// TwinCAT 3 PLC project Main
// ProgramVersion: 3.1.4026.22
// libraries:
//   mobject-core, * (mobject)
//   Tc2_Standard, * (Beckhoff Automation GmbH)
//   Tc2_System, * (Beckhoff Automation GmbH)
//   Tc2_Utilities, * (Beckhoff Automation GmbH)
//   Tc3_JsonXml, * (Beckhoff Automation GmbH)
//   Tc3_Module, * (Beckhoff Automation GmbH)
//   TcUnit, * (www.tcunit.org)
// project tree:
//   mobject-collections/ MobjectCollectionsExample.TcPOU, MobjectCollectionsUnitTests.TcPOU
//   mobject-collections/Tests/ DictionaryForwardEnumerator_TestSuite.TcPOU, DictionaryKeyValueForwardEnumerator_TestSuite.TcPOU (not stored), Dictionary_TestSuite.TcPOU (not stored), LinkedListForwardEnumerator_TestSuite.TcPOU, LinkedList_TestSuite.TcPOU, OrderedDicKeyValueForwardEnumerator_TestSuite.TcPOU, OrderedDictionaryForwardEnumerator_TestSuite.TcPOU (not stored), OrderedDictionary_TestSuite.TcPOU (not stored), QueueForwardEnumerator_TestSuite.TcPOU, Queue_TestSuite.TcPOU (not stored), StackForwardEnumerator_TestSuite.TcPOU (not stored), Stack_TestSuite.TcPOU
//   mobject-collections/Tests/Mocks/EventHandlers/ CollectionChangedEventHandler.TcPOU, CollectionDisposedEventHandler.TcPOU (not stored), CollectionEventHandler.TcPOU (not stored), CollectionEventHandlerBase.TcPOU, KeyValueCollectionChangedEventHandler.TcPOU (not stored), KeyValueCollectionDisposedEventHandler.TcPOU, KeyValueCollectionEventHandler.TcPOU
//   mobject-converters/ MobjectConvertersUnitTests.TcPOU
//   mobject-converters/Tests/ BOOL_TO_TestSuite.TcPOU (not stored), BYTE_TO_TestSuite.TcPOU, DATE_TO_TestSuite.TcPOU, DINT_TO_TestSuite.TcPOU, DT_TO_TestSuite.TcPOU (not stored), DWORD_TO_TestSuite.TcPOU (not stored), INT_TO_TestSuite.TcPOU, LINT_TO_TestSuite.TcPOU, LREAL_TO_TestSuite.TcPOU, LWORD_TO_TestSuite.TcPOU, REAL_TO_TestSuite.TcPOU, SINT_TO_TestSuite.TcPOU (not stored), STRING_TO_TestSuite.TcPOU, TIME_TO_TestSuite.TcPOU, TOD_TO_TestSuite.TcPOU, UDINT_TO_TestSuite.TcPOU, UINT_TO_TestSuite.TcPOU (not stored), ULINT_TO_TestSuite.TcPOU, USINT_TO_TestSuite.TcPOU, WORD_TO_TestSuite.TcPOU (not stored)
//   mobject-datatypes/ MobjectDatatypesUnitTests.TcPOU (not stored)
//   mobject-datatypes/Tests/ AliasDatatype_TestSuite.TcPOU (not stored), Datatype_TestSuite.TcPOU (not stored), EnumDatatype_TestSuite.TcPOU, StructuredDatatype_TestSuite.TcPOU (not stored), _ArrayDatatype_1D_TestSuite.TcPOU, _ArrayDatatype_2D_TestSuite.TcPOU, _ArrayDatatype_3D_TestSuite.TcPOU, _BIT_UsingMockStructure_TestSuite.TcPOU, _BOOL_TestSuite.TcPOU (not stored), _BYTE_TestSuite.TcPOU (not stored), _DINT_TestSuite.TcPOU, _DT_TestSuite.TcPOU (not stored), _DWORD_TestSuite.TcPOU (not stored), _INT_TestSuite.TcPOU (not stored), _LINT_TestSuite.TcPOU, _LREAL_TestSuite.TcPOU (not stored), _LWORD_TestSuite.TcPOU (not stored), _REAL_TestSuite.TcPOU, _SINT_TestSuite.TcPOU, _STRING_TestSuite.TcPOU (not stored), _TIME_OF_DAY_TestSuite.TcPOU (not stored), _TOD_TestSuite.TcPOU (not stored), _UDINT_TestSuite.TcPOU, _UINT_TestSuite.TcPOU, _ULINT_TestSuite.TcPOU, _USINT_TestSuite.TcPOU (not stored), _WORD_TestSuite.TcPOU (not stored)
//   mobject-datatypes/Tests/Mocks/1DimArray/ _Array0to10OfBool.TcPOU
//   mobject-datatypes/Tests/Mocks/2DimArray/ _Array0to1_0to2OfBool.TcPOU
//   mobject-datatypes/Tests/Mocks/3DimArray/ _Array0to1_0to2_0to3OfBool.TcPOU (not stored)
//   mobject-datatypes/Tests/Mocks/DUT/ MyStruct.TcDUT
//   mobject-datatypes/Tests/Mocks/ MockAliasDatatype_HRESULT.TcPOU, MockDatatype_BOOL.TcPOU (not stored), MockEnumDatatype_E_TcEventClass.TcPOU, MockStructuredDatatype_TIMESTRUCT.TcPOU, _MyStruct.TcPOU
//   mobject-deserialization/ MobjectDeserializationUnitTests.TcPOU (not stored)
//   mobject-deserialization/Tests/ CustomDeserializationFailedError_TestSuite.TcPOU, DeserializationErrorFactory_TestSuite.TcPOU, DeserializerGarbageCollector_TestSuite.TcPOU (not stored), IncorrectKeyTypeDeserializationError_TestSuite.TcPOU, IncorrectTypeDeserializationError_TestSuite.TcPOU, InvalidKeyDeserializationError_TestSuite.TcPOU, MissingKeyDeserializationError_TestSuite.TcPOU (not stored), InvalidArrayIndexDeserializationError_TestSuite.TcPOU (not stored)
//   mobject-deserialization/Tests/Mocks/ MockDisposableDeserializer.TcPOU
//   mobject-disposable/ MobjectDisposableUnitTests.TcPOU
//   mobject-disposable/Tests/ Disposable_TestSuite.TcPOU (not stored)
//   mobject-disposable/Tests/Mocks/ MockDisposable.TcPOU (not stored)
//   mobject-errors/ MobjectErrorsUnitTests.TcPOU
//   mobject-errors/Tests/ Error_TestSuite.TcPOU (not stored), NullError_TestSuite.TcPOU (not stored)
//   mobject-events/ MobjectEventsUnitTests.TcPOU
//   mobject-events/Tests/ EventEmitterInterface_TestSuite.TcPOU (not stored), EventEmitter_TestSuite.TcPOU (not stored), EventHandlerInterface_TestSuite.TcPOU (not stored), EventTargetInterface_TestSuite.TcPOU
//   mobject-events/Tests/Mocks/ MockEvent.TcPOU (not stored), MockEventHandler.TcPOU (not stored)
//   mobject-json/ MobjectJsonUnitTests.TcPOU
//   mobject-json/Tests/ JsonDeserializerArrayForwardEnumerator_TestSuite.TcPOU, JsonDeserializerObjectForwardEnumerator_TestSuite.TcPOU (not stored), JsonDeserializer_TestSuite.TcPOU, JsonDomParser_TestSuite.TcPOU, JsonSerializer_TestSuite.TcPOU
//   mobject-json/Tests/Mocks/ MockDeserializableUserObject.TcPOU, MockSerializableArray.TcPOU (not stored), MockSerializableUserObject.TcPOU
//   mobject-server/ MobjectServerUnitTests.TcPOU, Server_IntegrationTestSuite.TcPOU
//   mobject-server/Mocks/ AdjustableSizeReplyRpcHandler.TcPOU, RejectWithMessageAsyncHandler.TcPOU, RejectWithMessageSyncHandler.TcPOU, SyncToAsyncEchoRpcHandler.TcPOU
//   mobject-server/_Internal/ AsyncResponseSessionData_TestSuite.TcPOU, ChunkedRequestData_TestSuite.TcPOU
//   / PlcTask.TcTTO
//   Main/ MAIN.TcPOU
//   SharedMocks/ MockError.TcPOU, MockErrorVisitor.TcPOU (not stored), MockJsonSerializer.TcPOU
// real-time tasks:
//   TASK PlcTask: cycle T#10ms, priority 20, ADS port 350

CONFIGURATION Main
    RESOURCE PLC ON TwinCAT3
        TASK PlcTask(INTERVAL := T#10ms, PRIORITY := 20);
        PROGRAM MAIN WITH PlcTask : MAIN;
    END_RESOURCE
END_CONFIGURATION

// ---- mobject-datatypes/Tests/Mocks/DUT/MyStruct.TcDUT
TYPE MyStruct :
STRUCT
	MyBit : BIT;
END_STRUCT
END_TYPE

// ---- Main/MAIN.TcPOU
PROGRAM MAIN
VAR
END_VAR

// unit tests
MobjectCollectionsUnitTests();
MobjectConvertersUnitTests();
MobjectDatatypesUnitTests();
MobjectDeserializationUnitTests();
MobjectDisposableUnitTests();
MobjectErrorsUnitTests();
MobjectEventsUnitTests();
MobjectJsonUnitTests();
MobjectServerUnitTests();

// examples
MobjectCollectionsExample();

// tcunit
TcUnit.RUN();

END_PROGRAM

// ---- mobject-collections/MobjectCollectionsUnitTests.TcPOU
PROGRAM MobjectCollectionsUnitTests
VAR
	dictionary_TestSuite : Dictionary_TestSuite;
	dictionaryForwardEnumerator_TestSuite : DictionaryForwardEnumerator_TestSuite;
	dictionaryKeyValueForwardEnumerator_TestSuite : DictionaryKeyValueForwardEnumerator_TestSuite;
	orderedDictionary_TestSuite : OrderedDictionary_TestSuite;
	orderedDictionaryForwardEnumerator_TestSuite : OrderedDictionaryForwardEnumerator_TestSuite;
	orderedDicKeyValueForwardEnumerator_TestSuite : OrderedDicKeyValueForwardEnumerator_TestSuite;
    linkedList_TestSuite : LinkedList_TestSuite;
	linkedListForwardEnumerator_TestSuite : LinkedListForwardEnumerator_TestSuite;
	queue_TestSuite : Queue_TestSuite;
	queueForwardEnumerator_TestSuite : QueueForwardEnumerator_TestSuite;
    stack_TestSuite : Stack_TestSuite;
	stackForwardEnumerator_TestSuite : StackForwardEnumerator_TestSuite;
END_VAR

END_PROGRAM

// ---- mobject-collections/Tests/DictionaryForwardEnumerator_TestSuite.TcPOU
FUNCTION_BLOCK DictionaryForwardEnumerator_TestSuite EXTENDS TcUnit.FB_TestSuite
VAR
END_VAR

CheckIsValidAtStart();
CheckMoveNextReturnsFalseAtTheEnd();
CheckMoveNextReturnsTrueSingleItem();
CheckMoveNextReturnsFalseWhenEmpty();
CheckMoveNextReturnsTrueMultipleItems();
CheckReset();
CheckTryGet();
CheckTryGetTo();
CheckWorksWithArrays();
CheckWorksWithIntegers();
CheckWorksWithStrings();

METHOD PRIVATE CheckIsValidAtStart
VAR
	result : BOOL;
	dictionary : Dictionary;
	enumerator : I_ForwardEnumerator;
END_VAR
TEST('CheckIsValidAtStart');

enumerator := dictionary.GetEnumerator();

result := enumerator.IsValid;
enumerator.Dispose();

AssertTrue(
	Condition := result,
	Message := 'IsValid returned false'
);

TEST_FINISHED();
END_METHOD

METHOD PRIVATE CheckMoveNextReturnsFalseAtTheEnd
VAR
	in1 : INT := 123;
	result : BOOL;
	dictionary : Dictionary;
	enumerator : I_ForwardEnumerator;
END_VAR
TEST('CheckMoveNextReturnsFalseAtTheEnd');

dictionary.TryAdd('a',in1);
enumerator := dictionary.GetEnumerator();

enumerator.MoveNext();
result := enumerator.MoveNext();

enumerator.Dispose();

AssertFalse(result,
    'MoveNext did not correctly signal the end of the enumeration');
	
TEST_FINISHED();
END_METHOD

METHOD PRIVATE CheckMoveNextReturnsFalseWhenEmpty
VAR
	result : BOOL;
	dictionary : Dictionary;
	enumerator : I_ForwardEnumerator;
	count : DINT;
END_VAR
TEST('CheckMoveNextReturnsFalseWhenEmpty');

count := dictionary.Count;
enumerator := dictionary.GetEnumerator();

result := enumerator.MoveNext();
enumerator.Dispose();

AssertFalse(Condition := result,
    Message := 'MoveNext did not correctly signal the end of the enumeration');

TEST_FINISHED();
END_METHOD

METHOD PRIVATE CheckMoveNextReturnsTrueMultipleItems
VAR
	in1 : INT := 123;
	in2 : INT := 456;
	in3 : INT := 789;
	result : BOOL;
	dictionary : Dictionary;
	enumerator : I_ForwardEnumerator;
END_VAR
TEST('CheckMoveNextReturnsTrueMultipleItems');

dictionary.TryAdd('a',in1);
dictionary.TryAdd('b',in2);
dictionary.TryAdd('c',in3);
enumerator := dictionary.GetEnumerator();

result := enumerator.MoveNext();
enumerator.Dispose();

AssertTrue(result, 'MoveNext did not correctly signal there were more items to follow');

TEST_FINISHED();
END_METHOD

METHOD PRIVATE CheckMoveNextReturnsTrueSingleItem
VAR
	in1 : INT := 123;
	result : BOOL;
	dictionary : Dictionary;
	enumerator : I_ForwardEnumerator;
END_VAR
TEST('CheckMoveNextReturnsTrueSingleItem');

dictionary.TryAdd('a',in1);
enumerator := dictionary.GetEnumerator();

result := enumerator.MoveNext();
enumerator.Dispose();

AssertTrue(result,
    'MoveNext did not correctly signal there were more items to follow');
	
TEST_FINISHED();
END_METHOD

METHOD PRIVATE CheckReset
VAR
	in1 : ARRAY [0..1] OF REAL := [0.1,2.3];
	in2 : ARRAY [0..1] OF REAL := [1.2,3.4];
	in3 : ARRAY [0..1] OF REAL := [2.3,4.5];
	out : ARRAY [0..1] OF REAL;
	expected : ARRAY [0..1] OF REAL := [0.1,2.3];
	dictionary : Dictionary;
	enumerator : I_ForwardEnumerator;
END_VAR
TEST('CheckReset');

dictionary.TryAdd('a',in1);
dictionary.TryAdd('b',in2);
dictionary.TryAdd('c',in3);

enumerator := dictionary.GetEnumerator();

enumerator.MoveNext();
enumerator.MoveNext();
enumerator.Reset();
enumerator.MoveNext();
enumerator.TryGet(out);

enumerator.Dispose();

AssertEquals(
	Expected := expected,
	Actual := out,
	Message := 'Did not produce the expected result'
);

TEST_FINISHED();
END_METHOD

METHOD PRIVATE CheckTryGet
VAR
	in : INT := 123;
	out : INT;
	expected : INT := 123;
	result : BOOL;
	dictionary : Dictionary;
	enumerator : I_ForwardEnumerator;
END_VAR
TEST('CheckTryGet');

dictionary.TryAdd('a',in);
enumerator := dictionary.GetEnumerator();
enumerator.MoveNext();

result := enumerator.TryGet(out);
enumerator.Dispose();

AssertTrue(
	Condition := result,
	Message := 'Method returned false'
);

AssertEquals(
	Expected := expected,
	Actual := out,
	Message := 'Did not produce the expected result'
);

TEST_FINISHED();
END_METHOD

METHOD PRIVATE CheckTryGetTo
VAR
	in : INT := 123;
	out : INT;
	expected : INT := 123;
	result : BOOL;
	dictionary : Dictionary;
	enumerator : I_ForwardEnumerator;
END_VAR
TEST('CheckTryGetTo');

dictionary.TryAdd('a',in);
enumerator := dictionary.GetEnumerator();
enumerator.MoveNext();

result := enumerator.TryGetTo(ADR(out),SIZEOF(out));
enumerator.Dispose();

AssertTrue(
	Condition := result,
	Message := 'Method returned false'
);

AssertEquals(
	Expected := expected,
	Actual := out,
	Message := 'Did not produce the expected result'
);

TEST_FINISHED();
END_METHOD

METHOD PRIVATE CheckWorksWithArrays
VAR
	in1 : ARRAY [0..1] OF REAL := [0.1,2.3];
	in2 : ARRAY [0..1] OF REAL := [1.2,3.4];
	in3 : ARRAY [0..1] OF REAL := [2.3,4.5];
	out1 : ARRAY [0..1] OF REAL;
	out2 : ARRAY [0..1] OF REAL;
	out3 : ARRAY [0..1] OF REAL;
	expected1 : ARRAY [0..1] OF REAL := [0.1,2.3];
	expected2 : ARRAY [0..1] OF REAL := [1.2,3.4];
	expected3 : ARRAY [0..1] OF REAL := [2.3,4.5];
	dictionary : Dictionary;
	enumerator : I_ForwardEnumerator;
END_VAR
TEST('CheckWorksWithArrays');

dictionary.TryAdd('c',in3);
dictionary.TryAdd('b',in2);
dictionary.TryAdd('a',in1);

enumerator := dictionary.GetEnumerator();

enumerator.MoveNext();
enumerator.TryGet(out1);
enumerator.MoveNext();
enumerator.TryGet(out2);
enumerator.MoveNext();
enumerator.TryGet(out3);

enumerator.Dispose();

AssertEquals(
	Expected := expected1,
	Actual := out1,
	Message := 'Did not produce the expected 1st result'
);

AssertEquals(
	Expected := expected2,
	Actual := out2,
	Message := 'Did not produce the expected 2nd result'
);

AssertEquals(
	Expected := expected3,
	Actual := out3,
	Message := 'Did not produce the expected 3rd result'
);

TEST_FINISHED();
END_METHOD

METHOD PRIVATE CheckWorksWithIntegers
VAR
	in1 : INT := 123;
	in2 : INT := 234;
	in3 : INT := 345;
	out1 : INT;
	out2 : INT;
	out3 : INT;
	expected1 : INT := 123;
	expected2 : INT := 234;
	expected3 : INT := 345;
	dictionary : Dictionary;
	enumerator : I_ForwardEnumerator;
END_VAR
TEST('CheckWorksWithIntegers');

dictionary.TryAdd('c',in3);
dictionary.TryAdd('b',in2);
dictionary.TryAdd('a',in1);

enumerator := dictionary.GetEnumerator();

enumerator.MoveNext();
enumerator.TryGet(out1);
enumerator.MoveNext();
enumerator.TryGet(out2);
enumerator.MoveNext();
enumerator.TryGet(out3);

enumerator.Dispose();

AssertEquals(
	Expected := expected1,
	Actual := out1,
	Message := 'Did not produce the expected 1st result'
);

AssertEquals(
	Expected := expected2,
	Actual := out2,
	Message := 'Did not produce the expected 2nd result'
);

AssertEquals(
	Expected := expected3,
	Actual := out3,
	Message := 'Did not produce the expected 3rd result'
);

TEST_FINISHED();
END_METHOD

METHOD PRIVATE CheckWorksWithStrings
VAR
	in1 : STRING := 'test1';
	in2 : STRING := 'test2';
	in3 : STRING := 'test3';
	out1 : STRING;
	out2 : STRING;
	out3 : STRING;
	expected1 : STRING := 'test1';
	expected2 : STRING := 'test2';
	expected3 : STRING := 'test3';
	dictionary : Dictionary;
	enumerator : I_ForwardEnumerator;
END_VAR
TEST('CheckWorksWithStrings');

dictionary.TryAdd('c',in3);
dictionary.TryAdd('b',in2);
dictionary.TryAdd('a',in1);

enumerator := dictionary.GetEnumerator();

enumerator.MoveNext();
enumerator.TryGet(out1);
enumerator.MoveNext();
enumerator.TryGet(out2);
enumerator.MoveNext();
enumerator.TryGet(out3);

enumerator.Dispose();

AssertEquals(
	Expected := expected1,
	Actual := out1,
	Message := 'Did not produce the expected 1st result'
);

AssertEquals(
	Expected := expected2,
	Actual := out2,
	Message := 'Did not produce the expected 2nd result'
);

AssertEquals(
	Expected := expected3,
	Actual := out3,
	Message := 'Did not produce the expected 3rd result'
);

TEST_FINISHED();
END_METHOD

END_FUNCTION_BLOCK

// ---- mobject-collections/Tests/OrderedDicKeyValueForwardEnumerator_TestSuite.TcPOU
FUNCTION_BLOCK OrderedDicKeyValueForwardEnumerator_TestSuite EXTENDS TcUnit.FB_TestSuite
VAR
END_VAR

CheckIsValidAtStart();
CheckKey();
CheckMoveNextReturnsFalseAtTheEnd();
CheckMoveNextReturnsTrueSingleItem();
CheckMoveNextReturnsFalseWhenEmpty();
CheckMoveNextReturnsTrueMultipleItems();
CheckReset();
CheckTryGet();
CheckTryGetTo();
CheckWorksWithArrays();
CheckWorksWithIntegers();
CheckWorksWithStrings();

METHOD PRIVATE CheckIsValidAtStart
VAR
	result : BOOL;
	dictionary : OrderedDictionary;
	enumerator : I_KeyValueForwardEnumerator;
END_VAR
TEST('CheckIsValidAtStart');

enumerator := dictionary.GetKeyValueEnumerator();

result := enumerator.IsValid;
enumerator.Dispose();

AssertTrue(
	Condition := result,
	Message := 'IsValid returned false'
);

TEST_FINISHED();
END_METHOD

METHOD PRIVATE CheckKey
VAR
	in1 : STRING := 'test1';
	in2 : STRING := 'test2';
	in3 : STRING := 'test3';
	out1 : STRING;
	out2 : STRING;
	out3 : STRING;
	expected1 : STRING := 'a';
	expected2 : STRING := 'b';
	expected3 : STRING := 'c';
	dictionary : OrderedDictionary;
	enumerator : I_KeyValueForwardEnumerator;
END_VAR
TEST('CheckKey');

dictionary.TryAdd('a',in1);
dictionary.TryAdd('b',in2);
dictionary.TryAdd('c',in3);

enumerator := dictionary.GetKeyValueEnumerator();

enumerator.MoveNext();
out1 := enumerator.Key;
enumerator.MoveNext();
out2 := enumerator.Key;
enumerator.MoveNext();
out3 := enumerator.Key;

enumerator.Dispose();

AssertEquals(
	Expected := expected1,
	Actual := out1,
	Message := 'Did not produce the expected 1st key'
);

AssertEquals(
	Expected := expected2,
	Actual := out2,
	Message := 'Did not produce the expected 2nd key'
);

AssertEquals(
	Expected := expected3,
	Actual := out3,
	Message := 'Did not produce the expected 3rd key'
);

TEST_FINISHED();
END_METHOD

METHOD PRIVATE CheckMoveNextReturnsFalseAtTheEnd
VAR
	in1 : INT := 123;
	result : BOOL;
	dictionary : OrderedDictionary;
	enumerator : I_KeyValueForwardEnumerator;
END_VAR
TEST('CheckMoveNextReturnsFalseAtTheEnd');

dictionary.TryAdd('a',in1);
enumerator := dictionary.GetKeyValueEnumerator();

enumerator.MoveNext();
result := enumerator.MoveNext();

enumerator.Dispose();

AssertFalse(result,
    'MoveNext did not correctly signal the end of the enumeration');
	
TEST_FINISHED();
END_METHOD

METHOD PRIVATE CheckMoveNextReturnsFalseWhenEmpty
VAR
	result : BOOL;
	dictionary : OrderedDictionary;
	enumerator : I_KeyValueForwardEnumerator;
	count : DINT;
END_VAR
TEST('CheckMoveNextReturnsFalseWhenEmpty');

count := dictionary.Count;
enumerator := dictionary.GetKeyValueEnumerator();

result := enumerator.MoveNext();
enumerator.Dispose();

AssertFalse(Condition := result,
    Message := 'MoveNext did not correctly signal the end of the enumeration');

TEST_FINISHED();
END_METHOD

METHOD PRIVATE CheckMoveNextReturnsTrueMultipleItems
VAR
	in1 : INT := 123;
	in2 : INT := 456;
	in3 : INT := 789;
	result : BOOL;
	dictionary : OrderedDictionary;
	enumerator : I_KeyValueForwardEnumerator;
END_VAR
TEST('CheckMoveNextReturnsTrueMultipleItems');

dictionary.TryAdd('a',in1);
dictionary.TryAdd('b',in2);
dictionary.TryAdd('c',in3);
enumerator := dictionary.GetKeyValueEnumerator();

result := enumerator.MoveNext();
enumerator.Dispose();

AssertTrue(result, 'MoveNext did not correctly signal there were more items to follow');

TEST_FINISHED();
END_METHOD

METHOD PRIVATE CheckMoveNextReturnsTrueSingleItem
VAR
	in1 : INT := 123;
	result : BOOL;
	dictionary : OrderedDictionary;
	enumerator : I_KeyValueForwardEnumerator;
END_VAR
TEST('CheckMoveNextReturnsTrueSingleItem');

dictionary.TryAdd('a',in1);
enumerator := dictionary.GetKeyValueEnumerator();

result := enumerator.MoveNext();
enumerator.Dispose();

AssertTrue(result,
    'MoveNext did not correctly signal there were more items to follow');
	
TEST_FINISHED();
END_METHOD

METHOD PRIVATE CheckReset
VAR
	in1 : ARRAY [0..1] OF REAL := [0.1,2.3];
	in2 : ARRAY [0..1] OF REAL := [1.2,3.4];
	in3 : ARRAY [0..1] OF REAL := [2.3,4.5];
	out : ARRAY [0..1] OF REAL;
	expected : ARRAY [0..1] OF REAL := [0.1,2.3];
	dictionary : OrderedDictionary;
	enumerator : I_KeyValueForwardEnumerator;
END_VAR
TEST('CheckReset');

dictionary.TryAdd('a',in1);
dictionary.TryAdd('b',in2);
dictionary.TryAdd('c',in3);

enumerator := dictionary.GetKeyValueEnumerator();

enumerator.MoveNext();
enumerator.MoveNext();
enumerator.Reset();
enumerator.MoveNext();
enumerator.TryGet(out);

enumerator.Dispose();

AssertEquals(
	Expected := expected,
	Actual := out,
	Message := 'Did not produce the expected result'
);

TEST_FINISHED();
END_METHOD

METHOD PRIVATE CheckTryGet
VAR
	in : INT := 123;
	out : INT;
	expected : INT := 123;
	result : BOOL;
	dictionary : OrderedDictionary;
	enumerator : I_KeyValueForwardEnumerator;
END_VAR
TEST('CheckTryGet');

dictionary.TryAdd('a',in);
enumerator := dictionary.GetKeyValueEnumerator();
enumerator.MoveNext();

result := enumerator.TryGet(out);
enumerator.Dispose();

AssertTrue(
	Condition := result,
	Message := 'Method returned false'
);

AssertEquals(
	Expected := expected,
	Actual := out,
	Message := 'Did not produce the expected result'
);

TEST_FINISHED();
END_METHOD

METHOD PRIVATE CheckTryGetTo
VAR
	in : INT := 123;
	out : INT;
	expected : INT := 123;
	result : BOOL;
	dictionary : OrderedDictionary;
	enumerator : I_KeyValueForwardEnumerator;
END_VAR
TEST('CheckTryGetTo');

dictionary.TryAdd('a',in);
enumerator := dictionary.GetKeyValueEnumerator();
enumerator.MoveNext();

result := enumerator.TryGetTo(ADR(out),SIZEOF(out));
enumerator.Dispose();

AssertTrue(
	Condition := result,
	Message := 'Method returned false'
);

AssertEquals(
	Expected := expected,
	Actual := out,
	Message := 'Did not produce the expected result'
);

TEST_FINISHED();
END_METHOD

METHOD PRIVATE CheckWorksWithArrays
VAR
	in1 : ARRAY [0..1] OF REAL := [0.1,2.3];
	in2 : ARRAY [0..1] OF REAL := [1.2,3.4];
	in3 : ARRAY [0..1] OF REAL := [2.3,4.5];
	out1 : ARRAY [0..1] OF REAL;
	out2 : ARRAY [0..1] OF REAL;
	out3 : ARRAY [0..1] OF REAL;
	expected1 : ARRAY [0..1] OF REAL := [0.1,2.3];
	expected2 : ARRAY [0..1] OF REAL := [1.2,3.4];
	expected3 : ARRAY [0..1] OF REAL := [2.3,4.5];
	dictionary : OrderedDictionary;
	enumerator : I_KeyValueForwardEnumerator;
END_VAR
TEST('CheckWorksWithArrays');

dictionary.TryAdd('c',in1);
dictionary.TryAdd('b',in2);
dictionary.TryAdd('a',in3);

enumerator := dictionary.GetKeyValueEnumerator();

enumerator.MoveNext();
enumerator.TryGet(out1);
enumerator.MoveNext();
enumerator.TryGet(out2);
enumerator.MoveNext();
enumerator.TryGet(out3);

enumerator.Dispose();

AssertEquals(
	Expected := expected1,
	Actual := out1,
	Message := 'Did not produce the expected 1st result'
);

AssertEquals(
	Expected := expected2,
	Actual := out2,
	Message := 'Did not produce the expected 2nd result'
);

AssertEquals(
	Expected := expected3,
	Actual := out3,
	Message := 'Did not produce the expected 3rd result'
);

TEST_FINISHED();
END_METHOD

METHOD PRIVATE CheckWorksWithIntegers
VAR
	in1 : INT := 123;
	in2 : INT := 234;
	in3 : INT := 345;
	out1 : INT;
	out2 : INT;
	out3 : INT;
	expected1 : INT := 123;
	expected2 : INT := 234;
	expected3 : INT := 345;
	dictionary : OrderedDictionary;
	enumerator : I_KeyValueForwardEnumerator;
END_VAR
TEST('CheckWorksWithIntegers');

dictionary.TryAdd('c',in1);
dictionary.TryAdd('b',in2);
dictionary.TryAdd('a',in3);

enumerator := dictionary.GetKeyValueEnumerator();

enumerator.MoveNext();
enumerator.TryGet(out1);
enumerator.MoveNext();
enumerator.TryGet(out2);
enumerator.MoveNext();
enumerator.TryGet(out3);

enumerator.Dispose();

AssertEquals(
	Expected := expected1,
	Actual := out1,
	Message := 'Did not produce the expected 1st result'
);

AssertEquals(
	Expected := expected2,
	Actual := out2,
	Message := 'Did not produce the expected 2nd result'
);

AssertEquals(
	Expected := expected3,
	Actual := out3,
	Message := 'Did not produce the expected 3rd result'
);

TEST_FINISHED();
END_METHOD

METHOD PRIVATE CheckWorksWithStrings
VAR
	in1 : STRING := 'test1';
	in2 : STRING := 'test2';
	in3 : STRING := 'test3';
	out1 : STRING;
	out2 : STRING;
	out3 : STRING;
	expected1 : STRING := 'test1';
	expected2 : STRING := 'test2';
	expected3 : STRING := 'test3';
	dictionary : OrderedDictionary;
	enumerator : I_KeyValueForwardEnumerator;
END_VAR
TEST('CheckWorksWithStrings');

dictionary.TryAdd('c',in1);
dictionary.TryAdd('b',in2);
dictionary.TryAdd('a',in3);

enumerator := dictionary.GetKeyValueEnumerator();

enumerator.MoveNext();
enumerator.TryGet(out1);
enumerator.MoveNext();
enumerator.TryGet(out2);
enumerator.MoveNext();
enumerator.TryGet(out3);

enumerator.Dispose();

AssertEquals(
	Expected := expected1,
	Actual := out1,
	Message := 'Did not produce the expected 1st result'
);

AssertEquals(
	Expected := expected2,
	Actual := out2,
	Message := 'Did not produce the expected 2nd result'
);

AssertEquals(
	Expected := expected3,
	Actual := out3,
	Message := 'Did not produce the expected 3rd result'
);

TEST_FINISHED();
END_METHOD

END_FUNCTION_BLOCK

// ---- mobject-collections/Tests/LinkedList_TestSuite.TcPOU
FUNCTION_BLOCK PUBLIC LinkedList_TestSuite EXTENDS TcUnit.FB_TestSuite

// check datatypes are handled correctly
CheckListWorksWithIntegers();
CheckListWorksWithStrings();
CheckListWorksWithArrays();

// all other checks
CheckLinkedListImplementsI_LinkedList();
CheckFirstIsCorrectWithOneValue();
CheckFirstIsCorrectWithMultipleValues();
CheckLastIsCorrectWithOneValue();
CheckLastIsCorrectWithMultipleValues();
CheckAddAfter();
CheckAddBefore();
CheckAddFirst();
CheckAddItem();
CheckAddLast();
CheckClear();
CheckRemove();
CheckRemoveFirst();
CheckTryRemoveItem();
CheckRemoveLast();
CheckCount();
CheckFind();
CheckFindLast();
CheckLinkedListReturnsEnumerator();
CheckOnChangedEvent();
CheckOnDisposedEvent();
CheckOnceEvent();
CheckOffEvent();
CheckTryCopyTo();
CheckEnumeratorIsInvalidAfterChange();
CheckIsEmptyWhenEmpty();
CheckIsEmptyWhenFull();

METHOD PUBLIC CheckAddAfter
VAR
	in1 : INT := 123;
	in2 : INT := 456;
	in3 : INT := 789;
	out : INT;
	expected : INT := 789;
	linkedList : LinkedList;
END_VAR
TEST('CheckAddAfter');

// @TEST-FIXTURE
linkedList.AddFirst(in1); // (first->) 123 (<-last)
linkedList.AddFirst(in2); // (first->) 456, 123 (<-last)

// @TEST-RUN
linkedList.AddAfter(linkedList.Last, in3); // (first->) 456, 123, 789 (<-last)
linkedList.Last.TryGet(out);

// @TEST-ASSSERT
AssertEquals(
	Expected := expected,
	Actual := out,
	Message := 'Did not produce the expected result'
);

TEST_FINISHED();
END_METHOD

METHOD PUBLIC CheckAddBefore
VAR
	in1 : INT := 123;
	in2 : INT := 456;
	in3 : INT := 789;
	out : INT;
	expected : INT := 789;
	linkedList : LinkedList;
END_VAR
TEST('CheckAddBefore');

// @TEST-FIXTURE
linkedList.AddFirst(in1); // (first->) 123 (<-last)
linkedList.AddFirst(in2); // (first->) 456, 123 (<-last)

// @TEST-RUN
linkedList.AddBefore(linkedList.First, in3); // (first->) 789, 456, 123 (<-last)
linkedList.First.TryGet(out);

// @TEST-ASSSERT
AssertEquals(
	Expected := expected,
	Actual := out,
	Message := 'Did not produce the expected result'
);

TEST_FINISHED();
END_METHOD

METHOD PUBLIC CheckAddFirst
VAR
	in1 : INT := 123;
	in2 : INT := 456;
	in3 : INT := 789;
	out : INT;
	expected : INT := 789;
	linkedList : LinkedList;
END_VAR
TEST('CheckAddFirst');

// @TEST-FIXTURE
linkedList.AddLast(in1); // (first->) 123 (<-last)
linkedList.AddLast(in2); // (first->) 123, 456 (<-last)

// @TEST-RUN
linkedList.AddFirst(in3); // (first->) 789, 123, 456 (<-last)
linkedList.First.TryGet(out);

// @TEST-ASSSERT
AssertEquals(
	Expected := expected,
	Actual := out,
	Message := 'Did not produce the expected result'
);

TEST_FINISHED();
END_METHOD

METHOD PUBLIC CheckAddItem
VAR
	in1 : INT := 123;
	in2 : INT := 456;
	in3 : INT := 789;
	out : INT;
	expected : INT := 789;
	linkedList : LinkedList;
END_VAR
TEST('CheckAddItem');

// @TEST-FIXTURE
linkedList.AddFirst(in1); // (first->) 123 (<-last)
linkedList.AddFirst(in2); // (first->) 456, 123 (<-last)

// @TEST-RUN
linkedList.AddItem(in3); // (first->) 456, 123, 789 (<-last)
linkedList.Last.TryGet(out);

// @TEST-ASSSERT
AssertEquals(
	Expected := expected,
	Actual := out,
	Message := 'Did not produce the expected result'
);

TEST_FINISHED();
END_METHOD

METHOD PUBLIC CheckAddLast
VAR
	in1 : INT := 123;
	in2 : INT := 456;
	in3 : INT := 789;
	out : INT;
	expected : INT := 789;
	linkedList : LinkedList;
END_VAR
TEST('CheckAddLast');

// @TEST-FIXTURE
linkedList.AddFirst(in1); // (first->) 123 (<-last)
linkedList.AddFirst(in2); // (first->) 456, 123 (<-last)

// @TEST-RUN
linkedList.AddLast(in3); // (first->) 456, 123, 789 (<-last)
linkedList.Last.TryGet(out);

// @TEST-ASSSERT
AssertEquals(
	Expected := expected,
	Actual := out,
	Message := 'Did not produce the expected result'
);

TEST_FINISHED();
END_METHOD

METHOD PUBLIC CheckClear
VAR
	in1 : INT := 123;
	in2 : INT := 456;
	out : INT;
	expected : INT := 456;
	linkedList : LinkedList;
END_VAR
TEST('CheckClear');

// @TEST-FIXTURE
linkedList.AddFirst(in1); // (first->) 123 (<-last)

// @TEST-RUN
linkedList.Clear();
linkedList.AddFirst(in2); // (first->) 456 (<-last) // if clear did not work then it would have (first->) 456, 123 (<-last)
linkedList.Last.TryGet(out);

// @TEST-ASSSERT
AssertEquals(
	Expected := expected,
	Actual := out,
	Message := 'Did not produce the expected result'
);

TEST_FINISHED();
END_METHOD

METHOD PUBLIC CheckCount
VAR
	in1 : INT := 123;
	in2 : INT := 456;
	in3 : INT := 789;
	out : DINT;
	expected : DINT := 3;
	linkedList : LinkedList;
END_VAR
TEST('CheckCount');

// @TEST-FIXTURE
linkedList.AddFirst(in1);
linkedList.AddFirst(in2);
linkedList.AddFirst(in3);

// @TEST-RUN
out := linkedList.Count;

// @TEST-ASSSERT
AssertEquals(
	Expected := expected,
	Actual := out,
	Message := 'Did not produce the expected result'
);

TEST_FINISHED();
END_METHOD

METHOD PUBLIC CheckEnumeratorIsInvalidAfterChange
VAR
	in : INT := 123;
	result : BOOL;
	linkedList : LinkedList;
	enumerator : I_ForwardEnumerator;
END_VAR
TEST('CheckEnumeratorIsInvalidAfterChange');

// @TEST-FIXTURE
enumerator := linkedList.GetEnumerator();
linkedList.AddItem(in);

// @TEST-RUN
result := enumerator.IsValid;
enumerator.Dispose();

// @TEST-ASSSERT
AssertFalse(
	Condition := result,
	Message := 'Method returned true'
);

TEST_FINISHED();
END_METHOD

METHOD PUBLIC CheckFind
VAR
	in1 : INT := 123;
	in2 : INT := 456;
	foundNode : I_LinkedListNode;
	linkedList : LinkedList;
END_VAR
TEST('CheckFind');

// @TEST-FIXTURE
linkedList.AddFirst(in1); // (first->) 123 (<-last)
linkedList.AddFirst(in2); // (first->) 456, 123 (<-last)
linkedList.AddFirst(in1); // (first->) 123, 456, 123 (<-last)

// @TEST-RUN
foundNode := linkedList.Find(in1);

// @TEST-ASSSERT
AssertTrue(
	Condition := (foundNode = linkedList.First),
	Message := 'Did find the correct node'
);

TEST_FINISHED();
END_METHOD

METHOD PUBLIC CheckFindLast
VAR
	in1 : INT := 123;
	in2 : INT := 456;
	foundNode : I_LinkedListNode;
	linkedList : LinkedList;
END_VAR
TEST('CheckFindLast');

// @TEST-FIXTURE
linkedList.AddFirst(in1); // (first->) 123 (<-last)
linkedList.AddFirst(in2); // (first->) 456, 123 (<-last)
linkedList.AddFirst(in1); // (first->) 123, 456, 123 (<-last)

// @TEST-RUN
foundNode := linkedList.FindLast(in1);

// @TEST-ASSSERT
AssertTrue(
	Condition := (foundNode = linkedList.Last),
	Message := 'Did find the correct node'
);

TEST_FINISHED();
END_METHOD

METHOD PUBLIC CheckFirstIsCorrectWithMultipleValues
VAR
	in1 : INT := 123;
	in2 : INT := 456;
	in3 : INT := 789;
	out : INT;
	expected : INT := 789;
	linkedList : LinkedList;
END_VAR
TEST('CheckFirstIsCorrectWithMultipleValues');

// @TEST-FIXTURE
linkedList.AddFirst(in1); // (first->) 123 (<-last)
linkedList.AddFirst(in2); // (first->) 456, 123 (<-last)
linkedList.AddFirst(in3); // (first->) 789, 456, 123 (<-last)
linkedList.First.TryGet(out);

// @TEST-RUN

// @TEST-ASSSERT
AssertEquals(
	Expected := expected,
	Actual := out,
	Message := 'Did not produce the expected result'
);

TEST_FINISHED();
END_METHOD

METHOD PUBLIC CheckFirstIsCorrectWithOneValue
VAR
	in : INT := 123;
	out : INT;
	expected : INT := 123;
	linkedList : LinkedList;
END_VAR
TEST('CheckFirstIsCorrectWithOneValue');

// @TEST-FIXTURE
linkedList.AddFirst(in);
linkedList.First.TryGet(out);

// @TEST-RUN

// @TEST-ASSSERT
AssertEquals(
	Expected := expected,
	Actual := out,
	Message := 'Did not produce the expected result'
);

TEST_FINISHED();
END_METHOD

METHOD PUBLIC CheckIsEmptyWhenEmpty
VAR
	result : BOOL;
	linkedList : LinkedList;
END_VAR
TEST('CheckIsEmptyWhenEmpty');

// @TEST-RUN
result := linkedList.IsEmpty;

// @TEST-ASSSERT
AssertTrue(
	Condition := result,
	Message := 'Incorrect state of IsEmpty'
);

TEST_FINISHED();
END_METHOD

METHOD PUBLIC CheckIsEmptyWhenFull
VAR
	in : INT := 123;
	result : BOOL;
	linkedList : LinkedList;
END_VAR
TEST('CheckIsEmptyWhenFull');

// @TEST-FIXTURE
linkedList.AddItem(in);

// @TEST-RUN
result := linkedList.IsEmpty;

// @TEST-ASSSERT
AssertFalse(
	Condition := result,
	Message := 'Incorrect state of IsEmpty'
);

TEST_FINISHED();
END_METHOD

METHOD PUBLIC CheckLastIsCorrectWithMultipleValues
VAR
	in1 : INT := 123;
	in2 : INT := 456;
	in3 : INT := 789;
	out : INT;
	expected : INT := 123;
	linkedList : LinkedList;
END_VAR
TEST('CheckLastIsCorrectWithMultipleValues');

// @TEST-FIXTURE
linkedList.AddFirst(in1); // (first->) 123 (<-last)
linkedList.AddFirst(in2); // (first->) 456, 123 (<-last)
linkedList.AddFirst(in3); // (first->) 789, 456, 123 (<-last)
linkedList.Last.TryGet(out);

// @TEST-RUN

// @TEST-ASSSERT
AssertEquals(
	Expected := expected,
	Actual := out,
	Message := 'Did not produce the expected result'
);

TEST_FINISHED();
END_METHOD

METHOD PUBLIC CheckLastIsCorrectWithOneValue
VAR
	in : INT := 123;
	out : INT;
	expected : INT := 123;
	linkedList : LinkedList;
END_VAR
TEST('CheckLastIsCorrectWithOneValue');

// @TEST-FIXTURE
linkedList.AddFirst(in);
linkedList.Last.TryGet(out);

// @TEST-RUN

// @TEST-ASSSERT
AssertEquals(
	Expected := expected,
	Actual := out,
	Message := 'Did not produce the expected result'
);

TEST_FINISHED();
END_METHOD

METHOD PUBLIC CheckLinkedListImplementsI_LinkedList
VAR
	linkedList : LinkedList;
    iLinkedList : I_LinkedList := linkedList;
    result : BOOL;
END_VAR
TEST('CheckLinkedListImplementsI_LinkedList');

// @TEST-FIXTURE

// @TEST-RUN
result := iLinkedList <> 0;

// @TEST-ASSSERT
AssertTrue(
	Condition := result,
	Message := 'Did not implement I_LinkedList'
);

TEST_FINISHED();
END_METHOD

METHOD PUBLIC CheckLinkedListReturnsEnumerator
VAR
	in1 : INT := 123;
	in2 : INT := 456;
	in3 : INT := 789;
	enumerator : I_ForwardEnumerator;
	linkedList : LinkedList;
END_VAR
TEST('CheckLinkedListReturnsEnumerator');

// @TEST-FIXTURE
linkedList.AddFirst(in1); // (first->) 123 (<-last)
linkedList.AddFirst(in2); // (first->) 456, 123 (<-last)
linkedList.AddFirst(in3); // (first->) 789, 456, 123 (<-last)

// @TEST-RUN
enumerator := linkedList.GetEnumerator();

// @TEST-ASSSERT
AssertTrue(
	Condition := (enumerator <> 0),
	Message := 'Did not return an enumerator'
);

// @TEST-DISPOSE
enumerator.Dispose();

TEST_FINISHED();
END_METHOD

METHOD PUBLIC CheckListWorksWithArrays
VAR
	in : ARRAY [0..1] OF REAL := [0.1,2.3];
	out : ARRAY [0..1] OF REAL;
	expected : ARRAY [0..1] OF REAL := [0.1,2.3];
	linkedList : LinkedList;
END_VAR
TEST('CheckListWorksWithArrays');

// @TEST-FIXTURE
linkedList.AddFirst(in);
linkedList.First.TryGet(out);

// @TEST-RUN

// @TEST-ASSSERT
AssertEquals(
	Expected := expected,
	Actual := out,
	Message := 'Did not produce the expected result'
);

TEST_FINISHED();
END_METHOD

METHOD PUBLIC CheckListWorksWithIntegers
VAR
	in : INT := 123;
	out : INT;
	expected : INT := 123;
	linkedList : LinkedList;
END_VAR
TEST('CheckListWorksWithIntegers');

// @TEST-FIXTURE
linkedList.AddFirst(in);
linkedList.First.TryGet(out);

// @TEST-RUN

// @TEST-ASSSERT
AssertEquals(
	Expected := expected,
	Actual := out,
	Message := 'Did not produce the expected result'
);

TEST_FINISHED();
END_METHOD

METHOD PUBLIC CheckListWorksWithStrings
VAR
	in : STRING := 'test';
	out : STRING;
	expected : STRING := 'test';
	linkedList : LinkedList;
END_VAR
TEST('CheckListWorksWithStrings');

// @TEST-FIXTURE
linkedList.AddFirst(in);
linkedList.First.TryGet(out);

// @TEST-RUN

// @TEST-ASSSERT
AssertEquals(
	Expected := expected,
	Actual := out,
	Message := 'Did not produce the expected result'
);

TEST_FINISHED();
END_METHOD

METHOD PUBLIC CheckOffEvent
VAR
	value : INT := 123;
	linkedList : LinkedList;
	handler : CollectionChangedEventHandler(ExpectedOriginator := linkedList);
END_VAR
TEST('CheckOffEvent');

// @TEST-FIXTURE
linkedList.OnEvent('OnChanged',handler);
linkedList.OffEvent('OnChanged',handler);

// @TEST-RUN
linkedList.AddFirst(value);

// @TEST-ASSSERT
AssertFalse(
	Condition := handler.EventReceived,
	Message := 'OnceEvent emitted the OnChanged event more than once'
);

TEST_FINISHED();
END_METHOD

METHOD PUBLIC CheckOnceEvent
VAR
	value : INT := 123;
	linkedList : LinkedList;
	handler : CollectionChangedEventHandler(ExpectedOriginator := linkedList);
END_VAR
TEST('CheckOnceEvent');

// @TEST-FIXTURE
linkedList.OnceEvent('OnChanged',handler);
linkedList.AddFirst(value);
handler.Reset();

// @TEST-RUN
linkedList.AddFirst(value);

// @TEST-ASSSERT
AssertFalse(
	Condition := handler.EventReceived,
	Message := 'OnceEvent emitted the OnChanged event more than once'
);

TEST_FINISHED();
END_METHOD

METHOD PUBLIC CheckOnChangedEvent
VAR
	value : INT := 123;
	linkedList : LinkedList;
	handler : CollectionChangedEventHandler(ExpectedOriginator := linkedList);
END_VAR
TEST('CheckOnChangedEvent');

// @TEST-FIXTURE
linkedList.OnEvent('OnChanged', handler);

// @TEST-RUN
linkedList.AddFirst(value);

// @TEST-ASSSERT
AssertTrue(
	Condition := handler.EventReceived,
	Message := 'Did not emit the OnChanged event'
);

AssertTrue(
	Condition := handler.FromExpectedOriginator,
	Message := 'Did not include itself in the OnChanged event'
);

TEST_FINISHED();
END_METHOD

METHOD PUBLIC CheckOnDisposedEvent
VAR
	value : INT := 123;
	pLinkedList : POINTER TO LinkedList;
	handler : CollectionDisposedEventHandler(ExpectedOriginator := 0);
END_VAR
TEST('CheckOnDisposedEvent');

// @TEST-FIXTURE
pLinkedList := __NEW(LinkedList);
handler.SetExpectedOriginator(pLinkedList^);
pLinkedList^.OnEvent('OnDisposed', handler);

// @TEST-RUN
pLinkedList^.Dispose();

// @TEST-ASSSERT
AssertTrue(
	Condition := handler.EventReceived,
	Message := 'Did not emit the OnDisposed event'
);

AssertTrue(
	Condition := handler.FromExpectedOriginator,
	Message := 'Did not include itself in the OnDisposed event'
);

TEST_FINISHED();
END_METHOD

METHOD PUBLIC CheckRemove
VAR
	in1 : INT := 123;
	in2 : INT := 456;
	in3 : INT := 789;
	result : BOOL;
	linkedList : LinkedList;
END_VAR
TEST('CheckRemove');

// @TEST-FIXTURE
linkedList.AddFirst(in1); // (first->) 123 (<-last)
linkedList.AddFirst(in2); // (first->) 456, 123 (<-last)
linkedList.AddFirst(in3); // (first->) 789, 456, 123 (<-last)

// @TEST-RUN
linkedList.Remove(in2); // (first->) 789, 123 (<-last)
result := linkedList.Contains(in2);

// @TEST-ASSSERT
AssertFalse(
	Condition := result,
	Message := 'Method returned true'
);

TEST_FINISHED();
END_METHOD

METHOD PUBLIC CheckRemoveFirst
VAR
	in1 : INT := 123;
	in2 : INT := 456;
	in3 : INT := 789;
	out : INT;
	expected : INT := 456;
	linkedList : LinkedList;
END_VAR
TEST('CheckRemoveFirst');

// @TEST-FIXTURE
linkedList.AddFirst(in1); // (first->) 123 (<-last)
linkedList.AddFirst(in2); // (first->) 456, 123 (<-last)
linkedList.AddFirst(in3); // (first->) 789, 456, 123 (<-last)
linkedList.RemoveFirst(); // (first->) 456, 123 (<-last)
linkedList.First.TryGet(out);

// @TEST-RUN

// @TEST-ASSSERT
AssertEquals(
	Expected := expected,
	Actual := out,
	Message := 'Did not produce the expected result'
);

TEST_FINISHED();
END_METHOD

METHOD PUBLIC CheckRemoveLast
VAR
	in1 : INT := 123;
	in2 : INT := 456;
	in3 : INT := 789;
	out : INT;
	expected : INT := 456;
	linkedList : LinkedList;
END_VAR
TEST('CheckRemoveLast');

// @TEST-FIXTURE
linkedList.AddFirst(in1); // (first->) 123 (<-last)
linkedList.AddFirst(in2); // (first->) 456, 123 (<-last)
linkedList.AddFirst(in3); // (first->) 789, 456, 123 (<-last)
linkedList.RemoveLast(); // (first->) 789, 456 (<-last)
linkedList.Last.TryGet(out);

// @TEST-RUN

// @TEST-ASSSERT
AssertEquals(
	Expected := expected,
	Actual := out,
	Message := 'Did not produce the expected result'
);

TEST_FINISHED();
END_METHOD

METHOD PUBLIC CheckTryCopyTo
VAR
	in1 : INT := 123;
	in2 : INT := 456;
	in3 : INT := 789;
	out : ARRAY [0..2] OF INT;
	expected : ARRAY [0..2] OF INT := [789,456,123];
	linkedList : LinkedList;
END_VAR
TEST('CheckTryCopyTo');

// @TEST-FIXTURE
linkedList.AddFirst(in1); // (first->) 123 (<-last)
linkedList.AddFirst(in2); // (first->) 456, 123 (<-last)
linkedList.AddFirst(in3); // (first->) 789, 456, 123 (<-last)

// @TEST-RUN
linkedList.TryCopyTo(out);

// @TEST-ASSSERT
AssertEquals(
	Expected := expected,
	Actual := out,
	Message := 'Did not produce the expected result'
);

TEST_FINISHED();
END_METHOD

METHOD PUBLIC CheckTryCopyToLocation
VAR
	in1 : INT := 123;
	in2 : INT := 456;
	in3 : INT := 789;
	out : ARRAY [0..2] OF INT;
	expected : ARRAY [0..2] OF INT := [789,456,123];
	linkedList : LinkedList;
END_VAR
TEST('CheckTryCopyToLocation');

// @TEST-FIXTURE
linkedList.AddFirst(in1); // (first->) 123 (<-last)
linkedList.AddFirst(in2); // (first->) 456, 123 (<-last)
linkedList.AddFirst(in3); // (first->) 789, 456, 123 (<-last)

// @TEST-RUN
linkedList.TryCopyToLocation(ADR(out),SIZEOF(out));

// @TEST-ASSSERT
AssertEquals(
	Expected := expected,
	Actual := out,
	Message := 'Did not produce the expected result'
);

TEST_FINISHED();
END_METHOD

METHOD PUBLIC CheckTryRemoveItem
VAR
	in1 : INT := 123;
	in2 : INT := 456;
	in3 : INT := 789;
	result : BOOL;
	linkedList : LinkedList;
END_VAR
TEST('CheckTryRemoveItem');

// @TEST-FIXTURE
linkedList.AddFirst(in1); // (first->) 123 (<-last)
linkedList.AddFirst(in2); // (first->) 456, 123 (<-last)
linkedList.AddFirst(in3); // (first->) 789, 456, 123 (<-last)

// @TEST-RUN
linkedList.TryRemoveItem(in2); // (first->) 789, 123 (<-last)
result := linkedList.Contains(in2);

// @TEST-ASSSERT
AssertFalse(
	Condition := result,
	Message := 'Method returned true'
);

TEST_FINISHED();
END_METHOD

END_FUNCTION_BLOCK

// ---- mobject-collections/Tests/Mocks/EventHandlers/CollectionChangedEventHandler.TcPOU
FUNCTION_BLOCK CollectionChangedEventHandler EXTENDS CollectionEventHandler

METHOD PUBLIC HandleEvent
VAR_INPUT
	Event : I_Event;
END_VAR
VAR
	changedEvent : I_CollectionChangedEvent;
END_VAR
IF __QUERYINTERFACE(Event, changedEvent) THEN
	_eventReceived := TRUE;
	fromExpected := changedEvent.Target = expectedOriginator;
END_IF
END_METHOD

END_FUNCTION_BLOCK

// ---- mobject-collections/Tests/LinkedListForwardEnumerator_TestSuite.TcPOU
FUNCTION_BLOCK PUBLIC LinkedListForwardEnumerator_TestSuite EXTENDS TcUnit.FB_TestSuite

CheckIsValidAtStart();
CheckMoveNextReturnsFalseAtTheEnd();
CheckMoveNextReturnsFalseWhenEmpty();
CheckMoveNextReturnsTrueMultipleItems();
CheckMoveNextReturnsTrueSingleItem();
CheckReset();
CheckTryGet();
CheckTryGetTo();
CheckWorksWithIntegers();
CheckWorksWithStrings();
CheckWorksWithArrays();

METHOD PUBLIC CheckIsValidAtStart
VAR
	result : BOOL;
	linkedList : LinkedList;
	enumerator : I_ForwardEnumerator;
END_VAR
TEST('CheckIsValidAtStart');

enumerator := linkedList.GetEnumerator();

result := enumerator.IsValid;
enumerator.Dispose();

AssertTrue(
	Condition := result,
	Message := 'Method returned false'
);

TEST_FINISHED();
END_METHOD

METHOD PRIVATE CheckMoveNextReturnsFalseAtTheEnd
VAR
	in1 : INT := 123;
	result : BOOL;
	linkedList : LinkedList;
	enumerator : I_ForwardEnumerator;
END_VAR
TEST('CheckMoveNextReturnsFalseAtTheEnd');

linkedList.AddLast(in1);
enumerator := linkedList.GetEnumerator();

enumerator.MoveNext();
result := enumerator.MoveNext();
enumerator.Dispose();

AssertFalse(result,
    'MoveNext did not correctly signal the end of the enumeration');
	
TEST_FINISHED();
END_METHOD

METHOD PUBLIC CheckMoveNextReturnsFalseWhenEmpty
VAR
	result : BOOL;
	linkedList : LinkedList;
	enumerator : I_ForwardEnumerator;
END_VAR
TEST('CheckMoveNextReturnsFalseWhenEmpty');

enumerator := linkedList.GetEnumerator();

result := enumerator.MoveNext();
enumerator.Dispose();

AssertFalse(
	Condition := result,
	Message := 'MoveNext did not correctly signal the end of the enumeration'
);

TEST_FINISHED();
END_METHOD

METHOD PRIVATE CheckMoveNextReturnsTrueMultipleItems
VAR
	in1 : INT := 123;
	in2 : INT := 456;
	in3 : INT := 789;
	result : BOOL;
	linkedList : LinkedList;
	enumerator : I_ForwardEnumerator;
END_VAR
TEST('CheckMoveNextReturnsTrueMultipleItems');

linkedList.AddLast(in1);
linkedList.AddLast(in2);
linkedList.AddLast(in3);
enumerator := linkedList.GetEnumerator();

result := enumerator.MoveNext();
enumerator.Dispose();

AssertTrue(result, 'MoveNext did not correctly signal there were more items to follow');

TEST_FINISHED();
END_METHOD

METHOD PRIVATE CheckMoveNextReturnsTrueSingleItem
VAR
	in1 : INT := 123;
	result : BOOL;
	linkedList : LinkedList;
	enumerator : I_ForwardEnumerator;
END_VAR
TEST('CheckMoveNextReturnsTrueSingleItem');

linkedList.AddLast(in1);
enumerator := linkedList.GetEnumerator();

result := enumerator.MoveNext();
enumerator.Dispose();

AssertTrue(result,
    'MoveNext did not correctly signal there were more items to follow');
	
TEST_FINISHED();
END_METHOD

METHOD PUBLIC CheckReset
VAR
	in1 : ARRAY [0..1] OF REAL := [0.1,2.3];
	in2 : ARRAY [0..1] OF REAL := [1.2,3.4];
	in3 : ARRAY [0..1] OF REAL := [2.3,4.5];
	out : ARRAY [0..1] OF REAL;
	expected : ARRAY [0..1] OF REAL := [0.1,2.3];
	linkedList : LinkedList;
	enumerator : I_ForwardEnumerator;
END_VAR
TEST('CheckReset');

linkedList.AddLast(in1);
linkedList.AddLast(in2);
linkedList.AddLast(in3);

enumerator := linkedList.GetEnumerator();

enumerator.MoveNext();
enumerator.MoveNext();
enumerator.Reset();
enumerator.MoveNext();
enumerator.TryGet(out);

enumerator.Dispose();

AssertEquals(
	Expected := expected,
	Actual := out,
	Message := 'Did not produce the expected result'
);

TEST_FINISHED();
END_METHOD

METHOD PUBLIC CheckTryGet
VAR
	in : INT := 123;
	out : INT;
	expected : INT := 123;
	result : BOOL;
	linkedList : LinkedList;
	enumerator : I_ForwardEnumerator;
END_VAR
TEST('CheckTryGet');

linkedList.AddLast(in);
enumerator := linkedList.GetEnumerator();
enumerator.MoveNext();

result := enumerator.TryGet(out);
enumerator.Dispose();

AssertTrue(
	Condition := result,
	Message := 'Method returned false'
);

AssertEquals(
	Expected := expected,
	Actual := out,
	Message := 'Did not produce the expected result'
);

TEST_FINISHED();
END_METHOD

METHOD PUBLIC CheckTryGetTo
VAR
	in : INT := 123;
	out : INT;
	expected : INT := 123;
	result : BOOL;
	linkedList : LinkedList;
	enumerator : I_ForwardEnumerator;
END_VAR
TEST('CheckTryGetTo');

linkedList.AddLast(in);
enumerator := linkedList.GetEnumerator();
enumerator.MoveNext();

result := enumerator.TryGetTo(ADR(out),SIZEOF(out));
enumerator.Dispose();

AssertTrue(
	Condition := result,
	Message := 'Method returned false'
);

AssertEquals(
	Expected := expected,
	Actual := out,
	Message := 'Did not produce the expected result'
);

TEST_FINISHED();
END_METHOD

METHOD PUBLIC CheckWorksWithArrays
VAR
	in1 : ARRAY [0..1] OF REAL := [0.1,2.3];
	in2 : ARRAY [0..1] OF REAL := [1.2,3.4];
	in3 : ARRAY [0..1] OF REAL := [2.3,4.5];
	out1 : ARRAY [0..1] OF REAL;
	out2 : ARRAY [0..1] OF REAL;
	out3 : ARRAY [0..1] OF REAL;
	expected1 : ARRAY [0..1] OF REAL := [0.1,2.3];
	expected2 : ARRAY [0..1] OF REAL := [1.2,3.4];
	expected3 : ARRAY [0..1] OF REAL := [2.3,4.5];
	linkedList : LinkedList;
	enumerator : I_ForwardEnumerator;
END_VAR
TEST('CheckWorksWithArrays');

linkedList.AddLast(in1);
linkedList.AddLast(in2);
linkedList.AddLast(in3);

enumerator := linkedList.GetEnumerator();

enumerator.MoveNext();
enumerator.TryGet(out1);
enumerator.MoveNext();
enumerator.TryGet(out2);
enumerator.MoveNext();
enumerator.TryGet(out3);

enumerator.Dispose();

AssertEquals(
	Expected := expected1,
	Actual := out1,
	Message := 'Did not produce the expected 1st result'
);

AssertEquals(
	Expected := expected2,
	Actual := out2,
	Message := 'Did not produce the expected 2nd result'
);

AssertEquals(
	Expected := expected3,
	Actual := out3,
	Message := 'Did not produce the expected 3rd result'
);

TEST_FINISHED();
END_METHOD

METHOD PUBLIC CheckWorksWithIntegers
VAR
	in1 : INT := 123;
	in2 : INT := 234;
	in3 : INT := 345;
	out1 : INT;
	out2 : INT;
	out3 : INT;
	expected1 : INT := 123;
	expected2 : INT := 234;
	expected3 : INT := 345;
	linkedList : LinkedList;
	enumerator : I_ForwardEnumerator;
END_VAR
TEST('CheckWorksWithIntegers');

linkedList.AddLast(in1);
linkedList.AddLast(in2);
linkedList.AddLast(in3);

enumerator := linkedList.GetEnumerator();

enumerator.MoveNext();
enumerator.TryGet(out1);
enumerator.MoveNext();
enumerator.TryGet(out2);
enumerator.MoveNext();
enumerator.TryGet(out3);

enumerator.Dispose();

AssertEquals(
	Expected := expected1,
	Actual := out1,
	Message := 'Did not produce the expected 1st result'
);

AssertEquals(
	Expected := expected2,
	Actual := out2,
	Message := 'Did not produce the expected 2nd result'
);

AssertEquals(
	Expected := expected3,
	Actual := out3,
	Message := 'Did not produce the expected 3rd result'
);

TEST_FINISHED();
END_METHOD

METHOD PUBLIC CheckWorksWithStrings
VAR
	in1 : STRING := 'test1';
	in2 : STRING := 'test2';
	in3 : STRING := 'test3';
	out1 : STRING;
	out2 : STRING;
	out3 : STRING;
	expected1 : STRING := 'test1';
	expected2 : STRING := 'test2';
	expected3 : STRING := 'test3';
	linkedList : LinkedList;
	enumerator : I_ForwardEnumerator;
END_VAR
TEST('CheckWorksWithStrings');

linkedList.AddLast(in1);
linkedList.AddLast(in2);
linkedList.AddLast(in3);

enumerator := linkedList.GetEnumerator();

enumerator.MoveNext();
enumerator.TryGet(out1);
enumerator.MoveNext();
enumerator.TryGet(out2);
enumerator.MoveNext();
enumerator.TryGet(out3);

enumerator.Dispose();

AssertEquals(
	Expected := expected1,
	Actual := out1,
	Message := 'Did not produce the expected 1st result'
);

AssertEquals(
	Expected := expected2,
	Actual := out2,
	Message := 'Did not produce the expected 2nd result'
);

AssertEquals(
	Expected := expected3,
	Actual := out3,
	Message := 'Did not produce the expected 3rd result'
);

TEST_FINISHED();
END_METHOD

END_FUNCTION_BLOCK

// ---- mobject-collections/Tests/QueueForwardEnumerator_TestSuite.TcPOU
FUNCTION_BLOCK PUBLIC QueueForwardEnumerator_TestSuite EXTENDS TcUnit.FB_TestSuite

CheckIsValidAtStart();
CheckMoveNextReturnsFalseAtTheEnd();
CheckMoveNextReturnsFalseWhenEmpty();
CheckMoveNextReturnsTrueMultipleItems();
CheckMoveNextReturnsTrueSingleItem();
CheckReset();
CheckTryGet();
CheckTryGetTo();
CheckWorksWithIntegers();
CheckWorksWithStrings();
CheckWorksWithArrays();

METHOD PUBLIC CheckIsValidAtStart
VAR
	result : BOOL;
	queue : Queue;
	enumerator : I_ForwardEnumerator;
END_VAR
TEST('CheckIsValidAtStart');

enumerator := queue.GetEnumerator();

result := enumerator.IsValid;
enumerator.Dispose();

AssertTrue(
	Condition := result,
	Message := 'Method returned false'
);

TEST_FINISHED();
END_METHOD

METHOD PRIVATE CheckMoveNextReturnsFalseAtTheEnd
VAR
	in1 : INT := 123;
	result : BOOL;
	queue : Queue;
	enumerator : I_ForwardEnumerator;
END_VAR
TEST('CheckMoveNextReturnsFalseAtTheEnd');

queue.Enqueue(in1);
enumerator := queue.GetEnumerator();

enumerator.MoveNext();
result := enumerator.MoveNext();
enumerator.Dispose();

AssertFalse(result,
    'MoveNext did not correctly signal the end of the enumeration');
	
TEST_FINISHED();
END_METHOD

METHOD PUBLIC CheckMoveNextReturnsFalseWhenEmpty
VAR
	result : BOOL;
	queue : Queue;
	enumerator : I_ForwardEnumerator;
END_VAR
TEST('CheckMoveNextReturnsFalseWhenEmpty');

enumerator := queue.GetEnumerator();

result := enumerator.MoveNext();
enumerator.Dispose();

AssertFalse(
	Condition := result,
	Message := 'MoveNext did not correctly signal the end of the enumeration'
);

TEST_FINISHED();
END_METHOD

METHOD PRIVATE CheckMoveNextReturnsTrueMultipleItems
VAR
	in1 : INT := 123;
	in2 : INT := 456;
	in3 : INT := 789;
	result : BOOL;
	queue : Queue;
	enumerator : I_ForwardEnumerator;
END_VAR
TEST('CheckMoveNextReturnsTrueMultipleItems');

queue.Enqueue(in1);
queue.Enqueue(in2);
queue.Enqueue(in3);
enumerator := queue.GetEnumerator();

result := enumerator.MoveNext();
enumerator.Dispose();

AssertTrue(result, 'MoveNext did not correctly signal there were more items to follow');

TEST_FINISHED();
END_METHOD

METHOD PRIVATE CheckMoveNextReturnsTrueSingleItem
VAR
	in1 : INT := 123;
	result : BOOL;
	queue : Queue;
	enumerator : I_ForwardEnumerator;
END_VAR
TEST('CheckMoveNextReturnsTrueSingleItem');

queue.Enqueue(in1);
enumerator := queue.GetEnumerator();

result := enumerator.MoveNext();
enumerator.Dispose();

AssertTrue(result,
    'MoveNext did not correctly signal there were more items to follow');
	
TEST_FINISHED();
END_METHOD

METHOD PUBLIC CheckReset
VAR
	in1 : ARRAY [0..1] OF REAL := [0.1,2.3];
	in2 : ARRAY [0..1] OF REAL := [1.2,3.4];
	in3 : ARRAY [0..1] OF REAL := [2.3,4.5];
	out : ARRAY [0..1] OF REAL;
	expected : ARRAY [0..1] OF REAL := [0.1,2.3];
	queue : Queue;
	enumerator : I_ForwardEnumerator;
END_VAR
TEST('CheckReset');

queue.Enqueue(in1);
queue.Enqueue(in2);
queue.Enqueue(in3);

enumerator := queue.GetEnumerator();

enumerator.MoveNext();
enumerator.MoveNext();
enumerator.Reset();
enumerator.MoveNext();
enumerator.TryGet(out);

enumerator.Dispose();

AssertEquals(
	Expected := expected,
	Actual := out,
	Message := 'Did not produce the expected result'
);

TEST_FINISHED();
END_METHOD

METHOD PUBLIC CheckTryGet
VAR
	in : INT := 123;
	out : INT;
	expected : INT := 123;
	result : BOOL;
	queue : Queue;
	enumerator : I_ForwardEnumerator;
END_VAR
TEST('CheckTryGet');

queue.Enqueue(in);
enumerator := queue.GetEnumerator();
enumerator.MoveNext();

result := enumerator.TryGet(out);
enumerator.Dispose();

AssertTrue(
	Condition := result,
	Message := 'Method returned false'
);

AssertEquals(
	Expected := expected,
	Actual := out,
	Message := 'Did not produce the expected result'
);

TEST_FINISHED();
END_METHOD

METHOD PUBLIC CheckTryGetTo
VAR
	in : INT := 123;
	out : INT;
	expected : INT := 123;
	result : BOOL;
	queue : Queue;
	enumerator : I_ForwardEnumerator;
END_VAR
TEST('CheckTryGetTo');

queue.Enqueue(in);
enumerator := queue.GetEnumerator();
enumerator.MoveNext();

result := enumerator.TryGetTo(ADR(out),SIZEOF(out));
enumerator.Dispose();

AssertTrue(
	Condition := result,
	Message := 'Method returned false'
);

AssertEquals(
	Expected := expected,
	Actual := out,
	Message := 'Did not produce the expected result'
);

TEST_FINISHED();
END_METHOD

METHOD PUBLIC CheckWorksWithArrays
VAR
	in1 : ARRAY [0..1] OF REAL := [0.1,2.3];
	in2 : ARRAY [0..1] OF REAL := [1.2,3.4];
	in3 : ARRAY [0..1] OF REAL := [2.3,4.5];
	out1 : ARRAY [0..1] OF REAL;
	out2 : ARRAY [0..1] OF REAL;
	out3 : ARRAY [0..1] OF REAL;
	expected1 : ARRAY [0..1] OF REAL := [0.1,2.3];
	expected2 : ARRAY [0..1] OF REAL := [1.2,3.4];
	expected3 : ARRAY [0..1] OF REAL := [2.3,4.5];
	queue : Queue;
	enumerator : I_ForwardEnumerator;
END_VAR
TEST('CheckWorksWithArrays');

queue.Enqueue(in1);
queue.Enqueue(in2);
queue.Enqueue(in3);

enumerator := queue.GetEnumerator();

enumerator.MoveNext();
enumerator.TryGet(out1);
enumerator.MoveNext();
enumerator.TryGet(out2);
enumerator.MoveNext();
enumerator.TryGet(out3);

enumerator.Dispose();

AssertEquals(
	Expected := expected1,
	Actual := out1,
	Message := 'Did not produce the expected 1st result'
);

AssertEquals(
	Expected := expected2,
	Actual := out2,
	Message := 'Did not produce the expected 2nd result'
);

AssertEquals(
	Expected := expected3,
	Actual := out3,
	Message := 'Did not produce the expected 3rd result'
);

TEST_FINISHED();
END_METHOD

METHOD PUBLIC CheckWorksWithIntegers
VAR
	in1 : INT := 123;
	in2 : INT := 234;
	in3 : INT := 345;
	out1 : INT;
	out2 : INT;
	out3 : INT;
	expected1 : INT := 123;
	expected2 : INT := 234;
	expected3 : INT := 345;
	queue : Queue;
	enumerator : I_ForwardEnumerator;
END_VAR
TEST('CheckWorksWithIntegers');

queue.Enqueue(in1);
queue.Enqueue(in2);
queue.Enqueue(in3);

enumerator := queue.GetEnumerator();

enumerator.MoveNext();
enumerator.TryGet(out1);
enumerator.MoveNext();
enumerator.TryGet(out2);
enumerator.MoveNext();
enumerator.TryGet(out3);

enumerator.Dispose();

AssertEquals(
	Expected := expected1,
	Actual := out1,
	Message := 'Did not produce the expected 1st result'
);

AssertEquals(
	Expected := expected2,
	Actual := out2,
	Message := 'Did not produce the expected 2nd result'
);

AssertEquals(
	Expected := expected3,
	Actual := out3,
	Message := 'Did not produce the expected 3rd result'
);

TEST_FINISHED();
END_METHOD

METHOD PUBLIC CheckWorksWithStrings
VAR
	in1 : STRING := 'test1';
	in2 : STRING := 'test2';
	in3 : STRING := 'test3';
	out1 : STRING;
	out2 : STRING;
	out3 : STRING;
	expected1 : STRING := 'test1';
	expected2 : STRING := 'test2';
	expected3 : STRING := 'test3';
	queue : Queue;
	enumerator : I_ForwardEnumerator;
END_VAR
TEST('CheckWorksWithStrings');

queue.Enqueue(in1);
queue.Enqueue(in2);
queue.Enqueue(in3);

enumerator := queue.GetEnumerator();

enumerator.MoveNext();
enumerator.TryGet(out1);
enumerator.MoveNext();
enumerator.TryGet(out2);
enumerator.MoveNext();
enumerator.TryGet(out3);

enumerator.Dispose();

AssertEquals(
	Expected := expected1,
	Actual := out1,
	Message := 'Did not produce the expected 1st result'
);

AssertEquals(
	Expected := expected2,
	Actual := out2,
	Message := 'Did not produce the expected 2nd result'
);

AssertEquals(
	Expected := expected3,
	Actual := out3,
	Message := 'Did not produce the expected 3rd result'
);

TEST_FINISHED();
END_METHOD

END_FUNCTION_BLOCK

// ---- mobject-collections/Tests/Stack_TestSuite.TcPOU
FUNCTION_BLOCK PUBLIC Stack_TestSuite EXTENDS TcUnit.FB_TestSuite

// check datatypes are handled correctly
CheckListWorksWithIntegers();
CheckListWorksWithStrings();
CheckListWorksWithArrays();

// all other checks
CheckStackImplementsI_Stack();
CheckContains();
CheckClear();
CheckCount();
CheckAddItem();
CheckTryRemoveItem();
CheckTryPopRemovesTheItem();
CheckTryPopReturnsTheCorrectValue();
CheckTryPeekReturnsTheCorrectValue();
CheckTryPeekDoesNotRemoveTheItem();
CheckOnChangedEvent();
CheckOnDisposedEvent();
CheckOnceEvent();
CheckOffEvent();
CheckTryCopyTo();
CheckTryCopyToLocation();
CheckStackOrderIsCorrect();
CheckListReturnsEnumerator();
CheckEnumeratorIsInvalidAfterChange();
CheckIsEmptyWhenEmpty();
CheckIsEmptyWhenFull();

METHOD PUBLIC CheckAddItem
VAR
	in1 : INT := 123;
	in2 : INT := 456;
	in3 : INT := 789;
	result : BOOL;
	stack : Stack;
END_VAR
TEST('CheckAddItem');

// @TEST-FIXTURE
stack.Push(in1); // (fifo->) 123
stack.Push(in2); // (fifo->) 456, 123

// @TEST-RUN
stack.AddItem(in3); // fifo->) 789, 456, 123
result := stack.Contains(in3);

// @TEST-ASSSERT
AssertTrue(
	Condition := result,
	Message := 'Method returned false'
);

TEST_FINISHED();
END_METHOD

METHOD PUBLIC CheckClear
VAR
	in1 : INT := 123;
	in2 : INT := 456;
	in3 : INT := 789;
	stack : Stack;
END_VAR
TEST('CheckClear');

// @TEST-FIXTURE
stack.Push(in1); // (fifo->) 123
stack.Push(in2); // (fifo->) 456, 123
stack.Push(in2); // (fifo->) 789, 456, 123

// @TEST-RUN
stack.Clear();

// @TEST-ASSSERT
AssertTrue(
	Condition := stack.Count = 0,
	Message := 'The count is not zero'
);

TEST_FINISHED();
END_METHOD

METHOD PUBLIC CheckContains
VAR
	in1 : INT := 123;
	in2 : INT := 456;
	in3 : INT := 789;
	result : BOOL;
	stack : Stack;
END_VAR
TEST('CheckContains');

// @TEST-FIXTURE
stack.Push(in1); // (fifo->) 123
stack.Push(in2); // (fifo->) 456, 123
stack.Push(in2); // (fifo->) 789, 456, 123

// @TEST-RUN
result := stack.Contains(in2);

// @TEST-ASSSERT
AssertTrue(
	Condition := result,
	Message := 'Did not find the item in the queue'
);

TEST_FINISHED();
END_METHOD

METHOD PUBLIC CheckCount
VAR
	in1 : INT := 123;
	in2 : INT := 456;
	in3 : INT := 789;
	total : DINT;
	expected : DINT := 3;
	stack : Stack;
END_VAR
TEST('CheckCount');

// @TEST-FIXTURE
stack.Push(in1); // (fifo->) 123
stack.Push(in2); // (fifo->) 456, 123
stack.Push(in2); // (fifo->) 789, 456, 123

// @TEST-RUN
total := stack.Count;

// @TEST-ASSSERT
AssertEquals(
	Expected := expected,
	Actual := total,
	Message := 'Incorrect count'
);

TEST_FINISHED();
END_METHOD

METHOD PUBLIC CheckEnumeratorIsInvalidAfterChange
VAR
	in : INT := 123;
	result : BOOL;
	stack : Stack;
	enumerator : I_ForwardEnumerator;
END_VAR
TEST('CheckEnumeratorIsInvalidAfterChange');

// @TEST-FIXTURE
enumerator := stack.GetEnumerator();
stack.Push(in);

// @TEST-RUN
result := enumerator.IsValid;
enumerator.Dispose();

// @TEST-ASSSERT
AssertFalse(
	Condition := result,
	Message := 'Method returned true'
);

TEST_FINISHED();
END_METHOD

METHOD PUBLIC CheckIsEmptyWhenEmpty
VAR
	result : BOOL;
	stack : Stack;
END_VAR
TEST('CheckIsEmptyWhenEmpty');

// @TEST-RUN
result := stack.IsEmpty;

// @TEST-ASSSERT
AssertTrue(
	Condition := result,
	Message := 'Incorrect state of IsEmpty'
);

TEST_FINISHED();
END_METHOD

METHOD PUBLIC CheckIsEmptyWhenFull
VAR
	in : INT := 123;
	result : BOOL;
	stack : Stack;
END_VAR
TEST('CheckIsEmptyWhenFull');

// @TEST-FIXTURE
stack.Push(in);

// @TEST-RUN
result := stack.IsEmpty;

// @TEST-ASSSERT
AssertFalse(
	Condition := result,
	Message := 'Incorrect state of IsEmpty'
);

TEST_FINISHED();
END_METHOD

METHOD PUBLIC CheckListReturnsEnumerator
VAR
	in1 : INT := 123;
	in2 : INT := 456;
	in3 : INT := 789;
	enumerator : I_ForwardEnumerator;
	stack : Stack;
END_VAR
TEST('CheckListReturnsEnumerator');

// @TEST-FIXTURE
stack.Push(in1); // (fifo->) 123
stack.Push(in2); // (fifo->) 456, 123
stack.Push(in2); // (fifo->) 789, 456, 123

// @TEST-RUN
enumerator := stack.GetEnumerator();

// @TEST-ASSSERT
AssertTrue(
	Condition := (enumerator <> 0),
	Message := 'Did not return an enumerator'
);

// @TEST-DISPOSE
enumerator.Dispose();

TEST_FINISHED();
END_METHOD

METHOD PUBLIC CheckListWorksWithArrays
VAR
	in : ARRAY [0..1] OF REAL := [0.1,2.3];
	out : ARRAY [0..1] OF REAL;
	expected : ARRAY [0..1] OF REAL := [0.1,2.3];
	result : BOOL;
	stack : Stack;
END_VAR
TEST('CheckListWorksWithArrays');

// @TEST-FIXTURE
stack.Push(in);

// @TEST-RUN
result := stack.TryPop(out);

// @TEST-ASSSERT
AssertTrue(
	Condition := result,
	Message := 'Method returned false'
);

AssertEquals(
	Expected := expected,
	Actual := out,
	Message := 'Did not produce the expected result'
);

TEST_FINISHED();
END_METHOD

METHOD PUBLIC CheckListWorksWithIntegers
VAR
	in : INT := 123;
	out : INT;
	expected : INT := 123;
	result : BOOL;
	stack : Stack;
END_VAR
TEST('CheckListWorksWithIntegers');

// @TEST-FIXTURE
stack.Push(in);

// @TEST-RUN
result := stack.TryPop(out);

// @TEST-ASSSERT
AssertTrue(
	Condition := result,
	Message := 'Method returned false'
);

AssertEquals(
	Expected := expected,
	Actual := out,
	Message := 'Did not produce the expected result'
);

TEST_FINISHED();
END_METHOD

METHOD PUBLIC CheckListWorksWithStrings
VAR
	in : STRING := 'test';
	out : STRING;
	expected : STRING := 'test';
	result : BOOL;
	stack : Stack;
END_VAR
TEST('CheckListWorksWithStrings');

// @TEST-FIXTURE
stack.Push(in);

// @TEST-RUN
result := stack.TryPop(out);

// @TEST-ASSSERT
AssertTrue(
	Condition := result,
	Message := 'Method returned false'
);

AssertEquals(
	Expected := expected,
	Actual := out,
	Message := 'Did not produce the expected result'
);

TEST_FINISHED();
END_METHOD

METHOD PUBLIC CheckOffEvent
VAR
	value : INT := 123;
	stack : Stack;
	handler : CollectionChangedEventHandler(ExpectedOriginator := stack);
END_VAR
TEST('CheckOffEvent');

// @TEST-FIXTURE
stack.OnEvent('OnChanged',handler);
stack.OffEvent('OnChanged',handler);

// @TEST-RUN
stack.Push(value);

// @TEST-ASSSERT
AssertFalse(
	Condition := handler.EventReceived,
	Message := 'OnceEvent emitted the OnChanged event more than once'
);

TEST_FINISHED();
END_METHOD

METHOD PUBLIC CheckOnceEvent
VAR
	value : INT := 123;
	stack : Stack;
	handler : CollectionChangedEventHandler(ExpectedOriginator := stack);
END_VAR
TEST('CheckOnceEvent');

// @TEST-FIXTURE
stack.OnceEvent('OnChanged',handler);
stack.Push(value);
handler.Reset();

// @TEST-RUN
stack.Push(value);

// @TEST-ASSSERT
AssertFalse(
	Condition := handler.EventReceived,
	Message := 'OnceEvent emitted the OnChanged event more than once'
);

TEST_FINISHED();
END_METHOD

METHOD PUBLIC CheckOnChangedEvent
VAR
	value : INT := 123;
	stack : Stack;
	handler : CollectionChangedEventHandler(ExpectedOriginator := stack);
END_VAR
TEST('CheckOnChangedEvent');

// @TEST-FIXTURE
stack.OnEvent('OnChanged',handler);

// @TEST-RUN
stack.Push(value);

// @TEST-ASSSERT
AssertTrue(
	Condition := handler.EventReceived,
	Message := 'Did not emit the OnChanged event'
);

AssertTrue(
	Condition := handler.FromExpectedOriginator,
	Message := 'Did not include itself in the OnChanged event'
);

TEST_FINISHED();
END_METHOD

METHOD PUBLIC CheckOnDisposedEvent
VAR
	value : INT := 123;
	pStack : POINTER TO Stack;
	handler : CollectionDisposedEventHandler(ExpectedOriginator := 0);
END_VAR
TEST('CheckOnDisposedEvent');

// @TEST-FIXTURE
pStack := __NEW(Stack);
handler.SetExpectedOriginator(pStack^);
pStack^.OnEvent('OnDisposed',handler);

// @TEST-RUN
pStack^.Dispose();

// @TEST-ASSSERT
AssertTrue(
	Condition := handler.EventReceived,
	Message := 'Did not emit the OnDisposed event'
);

AssertTrue(
	Condition := handler.FromExpectedOriginator,
	Message := 'Did not include itself in the OnDisposed event'
);

TEST_FINISHED();
END_METHOD

METHOD PUBLIC CheckStackImplementsI_Stack
VAR
	stack : Stack;
    iStack : I_Stack := stack;
    result : BOOL;
END_VAR
TEST('CheckStackImplementsI_Stack');

// @TEST-FIXTURE

// @TEST-RUN
result := iStack <> 0;

// @TEST-ASSSERT
AssertTrue(
	Condition := result,
	Message := 'Did not implement I_Stack'
);

TEST_FINISHED();
END_METHOD

METHOD PUBLIC CheckStackOrderIsCorrect
VAR
	in1 : INT := 123;
	in2 : INT := 456;
	in3 : INT := 789;
	out1, out2, out3 : INT;
	expected1 : INT := 789;
	expected2 : INT := 456;
	expected3 : INT := 123;
	result1, result2, result3 : BOOL;
	stack : Stack;
END_VAR
TEST('CheckStackOrderIsCorrect');

// @TEST-FIXTURE
stack.Push(in1); // (fifo->) 123
stack.Push(in2); // (fifo->) 456, 123
stack.Push(in3); // (fifo->) 789, 456, 123

// @TEST-RUN
result1 := stack.TryPop(out1);
result2 := stack.TryPop(out2);
result3 := stack.TryPop(out3);

// @TEST-ASSSERT
AssertTrue(
	Condition := result1 AND result2 AND result3,
	Message := 'Method returned false'
);

AssertEquals(
	Expected := expected1,
	Actual := out1,
	Message := 'Did not produce the expected result'
);

AssertEquals(
	Expected := expected2,
	Actual := out2,
	Message := 'Did not produce the expected result'
);

AssertEquals(
	Expected := expected3,
	Actual := out3,
	Message := 'Did not produce the expected result'
);

TEST_FINISHED();
END_METHOD

METHOD PUBLIC CheckTryCopyTo
VAR
	in1 : INT := 123;
	in2 : INT := 456;
	in3 : INT := 789;
	out : ARRAY [0..2] OF INT;
	expected : ARRAY [0..2] OF INT := [789,456,123];
	stack : Stack;
END_VAR
TEST('CheckTryCopyTo');

// @TEST-FIXTURE
stack.Push(in1); // (fifo->) 123
stack.Push(in2); // (fifo->) 456, 123
stack.Push(in3); // (fifo->) 789, 456, 123

// @TEST-RUN
stack.TryCopyTo(out);

// @TEST-ASSSERT
AssertEquals(
	Expected := expected,
	Actual := out,
	Message := 'Did not produce the expected result'
);

TEST_FINISHED();
END_METHOD

METHOD PUBLIC CheckTryCopyToLocation
VAR
	in1 : INT := 123;
	in2 : INT := 456;
	in3 : INT := 789;
	out : ARRAY [0..2] OF INT;
	expected : ARRAY [0..2] OF INT := [789,456,123];
	stack : Stack;
END_VAR
TEST('CheckTryCopyToLocation');

// @TEST-FIXTURE
stack.Push(in1); // (fifo->) 123
stack.Push(in2); // (fifo->) 456, 123
stack.Push(in3); // (fifo->) 789, 456, 123

// @TEST-RUN
stack.TryCopyToLocation(ADR(out),SIZEOF(out));

// @TEST-ASSSERT
AssertEquals(
	Expected := expected,
	Actual := out,
	Message := 'Did not produce the expected result'
);

TEST_FINISHED();
END_METHOD

METHOD PUBLIC CheckTryPeekDoesNotRemoveTheItem
VAR
	in : INT := 123;
	out : INT;
	total : DINT;
	expected : DINT := 1;
	stack : Stack;
END_VAR
TEST('CheckTryPeekDoesNotRemoveTheItem');

// @TEST-FIXTURE
stack.Push(in); // (fifo->) 123

// @TEST-RUN
stack.TryPeek(out);
total := stack.Count;

// @TEST-ASSSERT
AssertEquals(
	Expected := expected,
	Actual := total,
	Message := 'Incorrect count'
);

TEST_FINISHED();
END_METHOD

METHOD PUBLIC CheckTryPeekReturnsTheCorrectValue
VAR
	in : INT := 123;
	out : INT;
	expected : INT := 123;
	result : BOOL;
	stack : Stack;
END_VAR
TEST('CheckTryPeekReturnsTheCorrectValue');

// @TEST-FIXTURE
stack.Push(in); // (fifo->) 123

// @TEST-RUN
result := stack.TryPeek(out);

// @TEST-ASSSERT
AssertTrue(
	Condition := result,
	Message := 'Method returned false'
);

AssertEquals(
	Expected := expected,
	Actual := out,
	Message := 'Did not produce the expected result'
);

TEST_FINISHED();
END_METHOD

METHOD PUBLIC CheckTryPopRemovesTheItem
VAR
	in : INT := 123;
	out : INT;
	total : DINT;
	expected : DINT := 0;
	stack : Stack;
END_VAR
TEST('CheckTryPopRemovesTheItem');

// @TEST-FIXTURE
stack.Push(in); // (fifo->) 123

// @TEST-RUN
stack.TryPop(out);
total := stack.Count;

// @TEST-ASSSERT
AssertEquals(
	Expected := expected,
	Actual := total,
	Message := 'Incorrect count'
);

TEST_FINISHED();
END_METHOD

METHOD PUBLIC CheckTryPopReturnsTheCorrectValue
VAR
	in : INT := 123;
	out : INT;
	expected : INT := 123;
	result : BOOL;
	stack : Stack;
END_VAR
TEST('CheckTryDequeueReturnsTheCorrectValue');

// @TEST-FIXTURE
stack.Push(in); // (fifo->) 123

// @TEST-RUN
result := stack.TryPop(out);

// @TEST-ASSSERT
AssertTrue(
	Condition := result,
	Message := 'Method returned false'
);

AssertEquals(
	Expected := expected,
	Actual := out,
	Message := 'Did not produce the expected result'
);

TEST_FINISHED();
END_METHOD

METHOD PUBLIC CheckTryRemoveItem
VAR
	in1 : INT := 123;
	in2 : INT := 456;
	in3 : INT := 789;
	result : BOOL;
	stack : Stack;
END_VAR
TEST('CheckTryRemoveItem');

// @TEST-FIXTURE
stack.Push(in1); // (fifo->) 123
stack.Push(in2); // (fifo->) 456, 123
stack.Push(in3); // (fifo->) 789, 456, 123

// @TEST-RUN
stack.TryRemoveItem(in2); // (lifo->) 789, 123
result := stack.Contains(in2);

// @TEST-ASSSERT
AssertFalse(
	Condition := result,
	Message := 'Method returned true'
);

TEST_FINISHED();
END_METHOD

END_FUNCTION_BLOCK

// ---- mobject-converters/MobjectConvertersUnitTests.TcPOU
PROGRAM MobjectConvertersUnitTests
VAR
	eventEmitter_TestSuite : EventEmitter_TestSuite;
	eventEmitterInterface_TestSuite : EventEmitterInterface_TestSuite;
	eventTargetInterface_TestSuite : EventTargetInterface_TestSuite;
	eventHandlerInterface_TestSuite : EventHandlerInterface_TestSuite;
END_VAR

END_PROGRAM

// ---- mobject-events/Tests/EventTargetInterface_TestSuite.TcPOU
FUNCTION_BLOCK PUBLIC EventTargetInterface_TestSuite EXTENDS TcUnit.FB_TestSuite
VAR
END_VAR

CheckEmitWorksWithHandler();
CheckExtendsFromQueryInterface();

METHOD PUBLIC CheckEmitWorksWithHandler
VAR
	mockEvent : MockEvent;
	mockHandler : MockEventHandler;
	eventEmitter : EventEmitter;
	iEventTarget : I_EventTarget := eventEmitter;
	eventReceived : BOOL;
END_VAR
TEST('CheckEmitWorksWithHandler');

eventEmitter.OnEvent('test', mockHandler);

iEventTarget.Emit('test',mockEvent);
eventReceived := mockHandler.EqualsLastEvent(mockEvent);

AssertTrue(
	Condition := eventReceived,
	Message := 'Event Emitter did not correctly emmit the event to the handler'
);

TEST_FINISHED();
END_METHOD

METHOD PUBLIC CheckExtendsFromQueryInterface
VAR
	eventEmitter : EventEmitter;
	iEventTarget : I_EventTarget := eventEmitter;
	iQueryInterface : __SYSTEM.IQueryInterface;
	result : BOOL;
END_VAR
TEST('CheckExtendsFromQueryInterface');

result := __QUERYINTERFACE(iEventTarget,iQueryInterface);

AssertTrue(
	Condition := result,
	Message := 'Interface did not extend __SYSTEM.IQueryInterface'
);

TEST_FINISHED();
END_METHOD

END_FUNCTION_BLOCK

// ---- mobject-disposable/MobjectDisposableUnitTests.TcPOU
PROGRAM MobjectDisposableUnitTests
VAR
	disposable_TestSuite : Disposable_TestSuite;
END_VAR

END_PROGRAM

// ---- mobject-errors/MobjectErrorsUnitTests.TcPOU
PROGRAM MobjectErrorsUnitTests
VAR
	error_TestSuite : Error_TestSuite;
	nullError_TestSuite : NullError_TestSuite;
END_VAR

END_PROGRAM

// ---- mobject-events/MobjectEventsUnitTests.TcPOU
PROGRAM MobjectEventsUnitTests
VAR
	eventEmitter_TestSuite : EventEmitter_TestSuite;
	eventEmitterInterface_TestSuite : EventEmitterInterface_TestSuite;
	eventTargetInterface_TestSuite : EventTargetInterface_TestSuite;
	eventHandlerInterface_TestSuite : EventHandlerInterface_TestSuite;
END_VAR

END_PROGRAM

// ---- mobject-json/MobjectJsonUnitTests.TcPOU
PROGRAM MobjectJsonUnitTests
VAR
	jsonDomParser_TestSuite : JsonDomParser_TestSuite;
	jsonSerializer_TestSuite : JsonSerializer_TestSuite;
	jsonDeserializer_TestSuite : JsonDeserializer_TestSuite;
	jsonDeserializerArrayForwardEnumerator_TestSuite : JsonDeserializerArrayForwardEnumerator_TestSuite;
	jsonDeserializerObjectForwardEnumerator_TestSuite : JsonDeserializerObjectForwardEnumerator_TestSuite;
END_VAR

END_PROGRAM

// ---- mobject-json/Tests/JsonDomParser_TestSuite.TcPOU
FUNCTION_BLOCK JsonDomParser_TestSuite EXTENDS TcUnit.FB_TestSuite
VAR
	jsonParser : JsonDomParser;
END_VAR

ModifyBoolArrayMemberFromJsonString();
ModifyDIntArrayMemberFromJsonString();
ModifyDIntPropertyFromJsonString();
ModifyFalseBoolPropertyFromJsonString();
ModifyIntArrayMemberFromJsonString();
ModifyIntPropertyFromJsonString();
ModifyLRealArrayMemberFromJsonString();
ModifyLRealPropertyFromJsonString();
ModifyRealArrayMemberFromJsonString();
ModifyRealPropertyFromJsonString();
ModifyStringPropertyFromJsonString();
ModifyTrueBoolPropertyFromJsonString();
ModifyUDIntArrayMemberFromJsonString();
ModifyUDIntPropertyFromJsonString();
ModifyValueFromChainedProperty();
ReadBoolArrayMemberFromJsonString();
ReadDIntArrayMemberFromJsonString();
ReadDIntPropertyFromJsonString();
ReadFalseBoolPropertyFromJsonString();
ReadIntArrayMemberFromJsonString();
ReadIntPropertyFromJsonString();
ReadLRealArrayMemberFromJsonString();
ReadLRealPropertyFromJsonString();
ReadRealArrayMemberFromJsonString();
ReadRealPropertyFromJsonString();
ReadStringPropertyFromJsonString();
ReadTrueBoolPropertyFromJsonString();
ReadUDIntArrayMemberFromJsonString();
ReadUDIntPropertyFromJsonString();
ReadValueFromChainedProperties();
TestTryLocateMethod();
TestTryWriteBoolMethod();
TestTryWriteDintMethod();
TestTryWriteIntMethod();
TestTryWriteLRealMethod();
TestTryWriteRealMethod();
TestTryWriteStringMethod();
TestTryWriteUdintMethod();

METHOD PUBLIC ModifyBoolArrayMemberFromJsonString
VAR_INPUT
END_VAR
VAR
	jsonTestString : T_MAXSTRING := '{"myArray" : [false, false, false]}';
	newValue : BOOL := TRUE;
	modifyResult : BOOL;
	result : BOOL;
	readResult : BOOL;
END_VAR
TEST('ModifyBoolArrayMemberFromJsonString');

// @TEST-RUN
jsonParser.ParseDocument(jsonTestString);
modifyResult := jsonParser.TryModify('.myArray[1]',newValue);
readResult := jsonParser.TryRead('.myArray[1]',result);
jsonParser.NewDocument();

// @TEST-ASSERT
AssertTrue(Condition := result, Message := 'Did not modify to the correct value');
AssertTrue(Condition := readResult, Message := 'Did not report a modify was successful');

TEST_FINISHED();
END_METHOD

METHOD PUBLIC ModifyDIntArrayMemberFromJsonString
VAR_INPUT
END_VAR
VAR
	jsonTestString : T_MAXSTRING := '{"myArray" : [123,456,789]}';
	newValue : DINT := 654;
	modifyResult : BOOL;
	actual : DINT;
	expected : DINT := 654;
	readResult : BOOL;
END_VAR
TEST('ModifyDIntArrayMemberFromJsonString');

// @TEST-RUN
jsonParser.ParseDocument(jsonTestString);
modifyResult := jsonParser.TryModify('.myArray[1]',newValue);
readResult := jsonParser.TryRead('.myArray[1]',actual);
jsonParser.NewDocument();

// @TEST-ASSERT
AssertEquals(Expected := expected, Actual := actual, Message := 'Did not modify to the correct value');
AssertTrue(Condition := modifyResult, Message := 'Did not report a modify was successful');

TEST_FINISHED();
END_METHOD

METHOD PUBLIC ModifyDIntPropertyFromJsonString
VAR_INPUT
END_VAR
VAR
	jsonTestString : T_MAXSTRING := '{"myDInt" : 123}';
	newValue : DINT := 456;
	modifyResult : BOOL;
	actual : DINT;
	expected : DINT := 456;
	readResult : BOOL;
END_VAR
TEST('ModifyDIntPropertyFromJsonString');

// @TEST-RUN
jsonParser.ParseDocument(jsonTestString);
modifyResult := jsonParser.TryModify('.myDInt',newValue);
readResult := jsonParser.TryRead('.myDInt',actual);
jsonParser.NewDocument();

// @TEST-ASSERT
AssertEquals(Expected := expected, Actual := actual, Message := 'Did not modify to the correct value');
AssertTrue(Condition := modifyResult, Message := 'Did not report a modify was successful');

TEST_FINISHED();
END_METHOD

METHOD PUBLIC ModifyFalseBoolPropertyFromJsonString
VAR_INPUT
END_VAR
VAR
	jsonTestString : T_MAXSTRING := '{"myTrueBool" : true, "myFalseBool" : false}';
	newValue : BOOL := TRUE;
	modifyResult : BOOL;
	result : BOOL;
	readResult : BOOL;
END_VAR
TEST('ModifyFalseBoolPropertyFromJsonString');

// @TEST-RUN
jsonParser.ParseDocument(jsonTestString);
modifyResult := jsonParser.TryModify('.myFalseBool',newValue);
readResult := jsonParser.TryRead('.myFalseBool',result);
jsonParser.NewDocument();

// @TEST-ASSERT
AssertTrue(Condition := result, Message := 'Did not modify to the correct value');
AssertTrue(Condition := modifyResult, Message := 'Did not report a modify was successful');

TEST_FINISHED();
END_METHOD

METHOD PUBLIC ModifyIntArrayMemberFromJsonString
VAR_INPUT
END_VAR
VAR
	jsonTestString : T_MAXSTRING := '{"myArray" : [123,456,789]}';
	newValue : INT := 654;
	modifyResult : BOOL;
	actual : INT;
	expected : INT := 654;
	readResult : BOOL;
END_VAR
TEST('ModifyIntArrayMemberFromJsonString');

// @TEST-RUN
jsonParser.ParseDocument(jsonTestString);
modifyResult := jsonParser.TryModify('.myArray[1]',newValue);
readResult := jsonParser.TryRead('.myArray[1]',actual);
jsonParser.NewDocument();

// @TEST-ASSERT
AssertEquals(Expected := expected, Actual := actual, Message := 'Did not modify to the correct value');
AssertTrue(Condition := modifyResult, Message := 'Did not report a modify was successful');

TEST_FINISHED();
END_METHOD

METHOD PUBLIC ModifyIntPropertyFromJsonString
VAR_INPUT
END_VAR
VAR
	jsonTestString : T_MAXSTRING := '{"myInt" : 123}';
	newValue : INT := 456;
	modifyResult : BOOL;
	actual : INT;
	expected : INT := 456;
	readResult : BOOL;
END_VAR
TEST('ModifyIntPropertyFromJsonString');

// @TEST-RUN
jsonParser.ParseDocument(jsonTestString);
modifyResult := jsonParser.TryModify('.myInt',newValue);
readResult := jsonParser.TryRead('.myInt',actual);
jsonParser.NewDocument();

// @TEST-ASSERT
AssertEquals(Expected := expected, Actual := actual, Message := 'Did not modify to the correct value');
AssertTrue(Condition := modifyResult, Message := 'Did not report a modify was successful');

TEST_FINISHED();
END_METHOD

METHOD PUBLIC ModifyLRealArrayMemberFromJsonString
VAR_INPUT
END_VAR
VAR
	jsonTestString : T_MAXSTRING := '{"myArray" : [123.1,456.2,789.3]}';
	newValue : LREAL := 678.4;
	modifyResult : BOOL;
	actual : LREAL;
	expected : LREAL := 678.4;
	readResult : BOOL;
END_VAR
TEST('ModifyLRealArrayMemberFromJsonString');

// @TEST-RUN
jsonParser.ParseDocument(jsonTestString);
modifyResult := jsonParser.TryModify('.myArray[1]',newValue);
readResult := jsonParser.TryRead('.myArray[1]',actual);
jsonParser.NewDocument();

// @TEST-ASSERT
AssertEquals(Expected := expected, Actual := actual, Message := 'Did not modify to the correct value');
AssertTrue(Condition := modifyResult, Message := 'Did not report a modify was successful');

TEST_FINISHED();
END_METHOD

METHOD PUBLIC ModifyLRealPropertyFromJsonString
VAR_INPUT
END_VAR
VAR
	jsonTestString : T_MAXSTRING := '{"myLReal" : 123.4}';
	newValue : LREAL := 456.5;
	modifyResult : BOOL;
	actual : LREAL;
	expected : LREAL := 456.5;
	readResult : BOOL;
END_VAR
TEST('ModifyLRealPropertyFromJsonString');

// @TEST-RUN
jsonParser.ParseDocument(jsonTestString);
modifyResult := jsonParser.TryModify('.myLReal',newValue);
readResult := jsonParser.TryRead('.myLReal',actual);
jsonParser.NewDocument();

// @TEST-ASSERT
AssertEquals(Expected := expected, Actual := actual, Message := 'Did not modify to the correct value');
AssertTrue(Condition := modifyResult, Message := 'Did not report a modify was successful');

TEST_FINISHED();
END_METHOD

METHOD PUBLIC ModifyRealArrayMemberFromJsonString
VAR_INPUT
END_VAR
VAR
	jsonTestString : T_MAXSTRING := '{"myArray" : [123.1,456.2,789.3]}';
	newValue : REAL := 678.4;
	modifyResult : BOOL;
	actual : REAL;
	expected : REAL := 678.4;
	readResult : BOOL;
END_VAR
TEST('ModifyRealArrayMemberFromJsonString');

// @TEST-RUN
jsonParser.ParseDocument(jsonTestString);
modifyResult := jsonParser.TryModify('.myArray[1]',newValue);
readResult := jsonParser.TryRead('.myArray[1]',actual);
jsonParser.NewDocument();

// @TEST-ASSERT
AssertEquals(Expected := expected, Actual := actual, Message := 'Did not modify to the correct value');
AssertTrue(Condition := modifyResult, Message := 'Did not report a modify was successful');

TEST_FINISHED();
END_METHOD

METHOD PUBLIC ModifyRealPropertyFromJsonString
VAR_INPUT
END_VAR
VAR
	jsonTestString : T_MAXSTRING := '{"myReal" : 123.4}';
	newValue : REAL := 456.5;
	modifyResult : BOOL;
	actual : REAL;
	expected : REAL := 456.5;
	readResult : BOOL;
END_VAR
TEST('ModifyRealPropertyFromJsonString');

// @TEST-RUN
jsonParser.ParseDocument(jsonTestString);
modifyResult := jsonParser.TryModify('.myReal',newValue);
readResult := jsonParser.TryRead('.myReal',actual);
jsonParser.NewDocument();

// @TEST-ASSERT
AssertEquals(Expected := expected, Actual := actual, Message := 'Did not modify to the correct value');
AssertTrue(Condition := modifyResult, Message := 'Did not report a modify was successful');

TEST_FINISHED();
END_METHOD

METHOD PUBLIC ModifyStringPropertyFromJsonString
VAR_INPUT
END_VAR
VAR
	jsonTestString : T_MAXSTRING := '{"myString" : "test"}';
	newValue : T_MAXSTRING := 'foobar';
	modifyResult : BOOL;
	actual : T_MAXSTRING;
	expected : T_MAXSTRING := 'foobar';
	readResult : BOOL;
END_VAR
TEST('ModifyStringPropertyFromJsonString');

// @TEST-RUN
jsonParser.ParseDocument(jsonTestString);
modifyResult := jsonParser.TryModify('.myString',newValue);
readResult := jsonParser.TryRead('.myString',actual);
jsonParser.NewDocument();

// @TEST-ASSERT
AssertEquals(Expected := expected, Actual := actual, Message := 'Did not modify to the correct value');
AssertTrue(Condition := modifyResult, Message := 'Did not report a modify was successful');

TEST_FINISHED();
END_METHOD

METHOD PUBLIC ModifyTrueBoolPropertyFromJsonString
VAR_INPUT
END_VAR
VAR
	jsonTestString : T_MAXSTRING := '{"myTrueBool" : true, "myFalseBool" : false}';
	newValue : BOOL := FALSE;
	modifyResult : BOOL;
	result : BOOL;
	readResult : BOOL;
END_VAR
TEST('ModifyTrueBoolPropertyFromJsonString');

// @TEST-RUN
jsonParser.ParseDocument(jsonTestString);
modifyResult := jsonParser.TryModify('.myTrueBool', newValue);
readResult := jsonParser.TryRead('.myTrueBool', result);
jsonParser.NewDocument();

// @TEST-ASSERT
AssertTrue(Condition := (result = newValue), Message := 'Did not modify to the correct value');
AssertTrue(Condition := modifyResult, Message := 'Did not report a modify was successful');

TEST_FINISHED();
END_METHOD

METHOD PUBLIC ModifyUDIntArrayMemberFromJsonString
VAR_INPUT
END_VAR
VAR
	jsonTestString : T_MAXSTRING := '{"myArray" : [123,456,789]}';
	newValue : UINT := 654;
	modifyResult : BOOL;
	actual : UINT;
	expected : UINT := 654;
	readResult : BOOL;
END_VAR
TEST('ModifyUDIntArrayMemberFromJsonString');

// @TEST-RUN
jsonParser.ParseDocument(jsonTestString);
modifyResult := jsonParser.TryModify('.myArray[1]',newValue);
readResult := jsonParser.TryRead('.myArray[1]',actual);
jsonParser.NewDocument();

// @TEST-ASSERT
AssertEquals(Expected := expected, Actual := actual, Message := 'Did not modify to the correct value');
AssertTrue(Condition := modifyResult, Message := 'Did not report a modify was successful');

TEST_FINISHED();
END_METHOD

METHOD PUBLIC ModifyUDIntPropertyFromJsonString
VAR_INPUT
END_VAR
VAR
	jsonTestString : T_MAXSTRING := '{"myUDInt" : 123}';
	newValue : UDINT := 456;
	modifyResult : BOOL;
	actual : UDINT;
	expected : UDINT := 456;
	readResult : BOOL;
END_VAR
TEST('ModifyUDIntPropertyFromJsonString');

// @TEST-RUN
jsonParser.ParseDocument(jsonTestString);
modifyResult := jsonParser.TryModify('.myUDInt',newValue);
readResult := jsonParser.TryRead('.myUDInt',actual);
jsonParser.NewDocument();

// @TEST-ASSERT
AssertEquals(Expected := expected, Actual := actual, Message := 'Did not modify to the correct value');
AssertTrue(Condition := modifyResult, Message := 'Did not report a modify was successful');

TEST_FINISHED();
END_METHOD

METHOD PUBLIC ModifyValueFromChainedProperty
VAR_INPUT
END_VAR
VAR
	jsonTestString : T_MAXSTRING := '{"level1" : {"level2" : {"level3" : {"level4" : 123}}}}';
	newValue : DINT := 456;
	modifyResult : BOOL;
	actual : DINT;
	expected : DINT := 456;
	readResult : BOOL;
END_VAR
TEST('ModifyValueFromChainedProperty');

// @TEST-RUN
jsonParser.ParseDocument(jsonTestString);
modifyResult := jsonParser.TryModify('.level1.level2.level3.level4',newValue);
readResult := jsonParser.TryRead('.level1.level2.level3.level4',actual);
jsonParser.NewDocument();

// @TEST-ASSERT
AssertEquals(Expected := expected, Actual := actual, Message := 'Did not modify to the correct value');
AssertTrue(Condition := modifyResult, Message := 'Did not report a modify was successful');

TEST_FINISHED();
END_METHOD

METHOD PUBLIC ReadBoolArrayMemberFromJsonString
VAR_INPUT
END_VAR
VAR
	jsonTestString : T_MAXSTRING := '{"myArray" : [false, true, false]}';
	result : BOOL;
	readResult : BOOL;
END_VAR
TEST('ReadBoolArrayMemberFromJsonString');

// @TEST-RUN
jsonParser.ParseDocument(jsonTestString);
readResult := jsonParser.TryRead('.myArray[1]',result);
jsonParser.NewDocument();

// @TEST-ASSERT
AssertTrue(Condition := result, Message := 'Did not read the correct value');
AssertTrue(Condition := readResult, Message := 'Did not report a read was successful');

TEST_FINISHED();
END_METHOD

METHOD PUBLIC ReadDIntArrayMemberFromJsonString
VAR_INPUT
END_VAR
VAR
	jsonTestString : T_MAXSTRING := '{"myArray" : [123,456,789]}';
	actual : DINT;
	expected : DINT := 456;
	readResult : BOOL;
END_VAR
TEST('ReadDIntArrayMemberFromJsonString');

// @TEST-RUN
jsonParser.ParseDocument(jsonTestString);
readResult := jsonParser.TryRead('.myArray[1]',Actual);
jsonParser.NewDocument();

// @TEST-ASSERT
AssertEquals(Expected := expected, Actual := actual, Message := 'Did not read the correct value');
AssertTrue(Condition := readResult, Message := 'Did not report a read was successful');

TEST_FINISHED();
END_METHOD

METHOD PUBLIC ReadDIntPropertyFromJsonString
VAR_INPUT
END_VAR
VAR
	jsonTestString : T_MAXSTRING := '{"myDInt" : 123}';
	actual : DINT;
	expected : DINT := 123;
	readResult : BOOL;
END_VAR
TEST('ReadDIntPropertyFromJsonString');

// @TEST-RUN
jsonParser.ParseDocument(jsonTestString);
readResult := jsonParser.TryRead('.myDInt',Actual);
jsonParser.NewDocument();

// @TEST-ASSERT
AssertEquals(Expected := expected, Actual := actual, Message := 'Did not read the correct value');
AssertTrue(Condition := readResult, Message := 'Did not report a read was successful');

TEST_FINISHED();
END_METHOD

METHOD PUBLIC ReadFalseBoolPropertyFromJsonString
VAR_INPUT
END_VAR
VAR
	jsonTestString : T_MAXSTRING := '{"myTrueBool" : true, "myFalseBool" : false}';
	result : BOOL;
	readResult : BOOL;
END_VAR
TEST('ReadFalseBoolPropertyFromJsonString');

// @TEST-RUN
jsonParser.ParseDocument(jsonTestString);
readResult := jsonParser.TryRead('.myFalseBool',result);
jsonParser.NewDocument();

// @TEST-ASSERT
AssertFalse(Condition := result, Message := 'Did not read the correct value');
AssertTrue(Condition := readResult, Message := 'Did not report a read was successful');

TEST_FINISHED();
END_METHOD

METHOD PUBLIC ReadIntArrayMemberFromJsonString
VAR_INPUT
END_VAR
VAR
	jsonTestString : T_MAXSTRING := '{"myArray" : [123,456,789]}';
	actual : INT;
	expected : INT := 456;
	readResult : BOOL;
END_VAR
TEST('ReadIntArrayMemberFromJsonString');

// @TEST-RUN
jsonParser.ParseDocument(jsonTestString);
readResult := jsonParser.TryRead('.myArray[1]',actual);
jsonParser.NewDocument();

// @TEST-ASSERT
AssertEquals(Expected := expected, Actual := actual, Message := 'Did not read the correct value');
AssertTrue(Condition := readResult, Message := 'Did not report a read was successful');

TEST_FINISHED();
END_METHOD

METHOD PUBLIC ReadIntPropertyFromJsonString
VAR_INPUT
END_VAR
VAR
	jsonTestString : T_MAXSTRING := '{"myInt" : 123}';
	actual : INT;
	expected : INT := 123;
	readResult : BOOL;
END_VAR
TEST('ReadIntPropertyFromJsonString');

// @TEST-RUN
jsonParser.ParseDocument(jsonTestString);
readResult := jsonParser.TryRead('.myInt',actual);
jsonParser.NewDocument();

// @TEST-ASSERT
AssertEquals(Expected := expected, Actual := actual, Message := 'Did not read the correct value');
AssertTrue(Condition := readResult, Message := 'Did not report a read was successful');

TEST_FINISHED();
END_METHOD

METHOD PUBLIC ReadLRealArrayMemberFromJsonString
VAR_INPUT
END_VAR
VAR
	jsonTestString : T_MAXSTRING := '{"myArray" : [-123.1,-456.2]}';
	actual : LREAL;
	expected : LREAL := -456.2;
	readResult : BOOL;
END_VAR
TEST('ReadLRealArrayMemberFromJsonString');

// @TEST-RUN
jsonParser.ParseDocument(jsonTestString);
readResult := jsonParser.TryRead('.myArray[1]',actual);
jsonParser.NewDocument();

// @TEST-ASSERT
AssertEquals(Expected := expected, Actual := actual, Message := 'Did not read the correct value');
AssertTrue(Condition := readResult, Message := 'Did not report a read was successful');

TEST_FINISHED();
END_METHOD

METHOD PUBLIC ReadLRealPropertyFromJsonString
VAR_INPUT
END_VAR
VAR
	jsonTestString : T_MAXSTRING := '{"myLReal" : -123.1}';
	actual : LREAL;
	expected : LREAL := -123.1;
	readResult : BOOL;
END_VAR
TEST('ReadLRealPropertyFromJsonString');

// @TEST-RUN
jsonParser.ParseDocument(jsonTestString);
readResult := jsonParser.TryRead('.myLReal',actual);
jsonParser.NewDocument();

// @TEST-ASSERT
AssertEquals(Expected := expected, Actual := actual, Message := 'Did not read the correct value');
AssertTrue(Condition := readResult, Message := 'Did not report a read was successful');

TEST_FINISHED();
END_METHOD

METHOD PUBLIC ReadRealArrayMemberFromJsonString
VAR_INPUT
END_VAR
VAR
	jsonTestString : T_MAXSTRING := '{"myArray" : [123.1,456.2,789.3]}';
	actual : REAL;
	expected : REAL := 456.2;
	readResult : BOOL;
END_VAR
TEST('ReadRealArrayMemberFromJsonString');

// @TEST-RUN
jsonParser.ParseDocument(jsonTestString);
readResult := jsonParser.TryRead('.myArray[1]',actual);
jsonParser.NewDocument();

// @TEST-ASSERT
AssertEquals(Expected := expected, Actual := actual, Message := 'Did not read the correct value');
AssertTrue(Condition := readResult, Message := 'Did not report a read was successful');

TEST_FINISHED();
END_METHOD

METHOD PUBLIC ReadRealPropertyFromJsonString
VAR_INPUT
END_VAR
VAR
	jsonTestString : T_MAXSTRING := '{"myReal" : 123.1}';
	actual : REAL;
	expected : REAL := 123.1;
	readResult : BOOL;
END_VAR
TEST('ReadRealPropertyFromJsonString');

// @TEST-RUN
jsonParser.ParseDocument(jsonTestString);
readResult := jsonParser.TryRead('.myReal',actual);
jsonParser.NewDocument();

// @TEST-ASSERT
AssertEquals(Expected := expected, Actual := actual, Message := 'Did not read the correct value');
AssertTrue(Condition := readResult, Message := 'Did not report a read was successful');

TEST_FINISHED();
END_METHOD

METHOD PUBLIC ReadStringPropertyFromJsonString
VAR_INPUT
END_VAR
VAR
	jsonTestString : T_MAXSTRING := '{"myString" : "test"}';
	actual : T_MAXSTRING;
	expected : T_MAXSTRING := 'test';
	readResult : BOOL;
END_VAR
TEST('ReadStringPropertyFromJsonString');

// @TEST-RUN
jsonParser.ParseDocument(jsonTestString);
readResult := jsonParser.TryRead('.myString',actual);
jsonParser.NewDocument();

// @TEST-ASSERT
AssertEquals(Expected := expected, Actual := actual, Message := 'Did not read the correct value');
AssertTrue(Condition := readResult, Message := 'Did not report a read was successful');

TEST_FINISHED();
END_METHOD

METHOD PUBLIC ReadTrueBoolPropertyFromJsonString
VAR_INPUT
END_VAR
VAR
	jsonTestString : T_MAXSTRING := '{"myTrueBool" : true, "myFalseBool" : false}';
	result : BOOL;
	readResult : BOOL;
END_VAR
TEST('ReadTrueBoolPropertyFromJsonString');

// @TEST-RUN
jsonParser.ParseDocument(jsonTestString);
readResult := jsonParser.TryRead('.myTrueBool',result);
jsonParser.NewDocument();

// @TEST-ASSERT
AssertTrue(Condition := result, Message := 'Did not read the correct value');
AssertTrue(Condition := readResult, Message := 'Did not report a read was successful');

TEST_FINISHED();
END_METHOD

METHOD PUBLIC ReadUDIntArrayMemberFromJsonString
VAR_INPUT
END_VAR
VAR
	jsonTestString : T_MAXSTRING := '{"myArray" : [123,456,789]}';
	actual : UDINT;
	expected : UDINT := 456;
	readResult : BOOL;
END_VAR
TEST('ReadUDIntArrayMemberFromJsonString');

// @TEST-RUN
jsonParser.ParseDocument(jsonTestString);
readResult := jsonParser.TryRead('.myArray[1]',actual);
jsonParser.NewDocument();

// @TEST-ASSERT
AssertEquals(Expected := expected, Actual := actual, Message := 'Did not read the correct value');
AssertTrue(Condition := readResult, Message := 'Did not report a read was successful');

TEST_FINISHED();
END_METHOD

METHOD PUBLIC ReadUDIntPropertyFromJsonString
VAR_INPUT
END_VAR
VAR
	jsonTestString : T_MAXSTRING := '{"myUDInt" : 123}';
	actual : UDINT;
	expected : UDINT := 123;
	readResult : BOOL;
END_VAR
TEST('ReadUDIntPropertyFromJsonString');

// @TEST-RUN
jsonParser.ParseDocument(jsonTestString);
readResult := jsonParser.TryRead('.myUDInt',actual);
jsonParser.NewDocument();

// @TEST-ASSERT
AssertEquals(Expected := expected, Actual := actual, Message := 'Did not read the correct value');
AssertTrue(Condition := readResult, Message := 'Did not report a read was successful');

TEST_FINISHED();
END_METHOD

METHOD PUBLIC ReadValueFromChainedProperties
VAR_INPUT
END_VAR
VAR
	jsonTestString : T_MAXSTRING := '{"level1" : {"level2" : {"level3" : {"level4" : 123}}}}';
	actual : DINT;
	expected : DINT := 123;
	readResult : BOOL;
END_VAR
TEST('ReadValueFromChainedProperties');

// @TEST-RUN
jsonParser.ParseDocument(jsonTestString);
readResult := jsonParser.TryRead('.level1.level2.level3.level4',actual);
jsonParser.NewDocument();

// @TEST-ASSERT
AssertEquals(Expected := expected, Actual := actual, Message := 'Did not read the correct value');
AssertTrue(Condition := readResult, Message := 'Did not report a read was successful');

TEST_FINISHED();
END_METHOD

METHOD PUBLIC TestTryLocateMethod
VAR_INPUT
END_VAR
VAR
	jsonTestString : T_MAXSTRING := '{"level1" : {"level2" : "test"}}';
	root : SJsonValue;
	level1 : SJsonValue;
	level2 : SJsonValue;
	actual : SJsonValue;
	locateResult : BOOL;
END_VAR
TEST('TestTryLocateMethod');

// @TEST-RUN
root := jsonParser.ParseDocument(jsonTestString);

// manually obtain the correct result
level1 := jsonParser.FindMember(root,'level1');
level2 := jsonParser.FindMember(level1,'level2');

locateResult := jsonParser.TryLocate('.level1.level2',actual);
jsonParser.NewDocument();

// @TEST-ASSERT
AssertEquals(Expected := level2, Actual := actual, Message := 'Did not locate the correct member');
AssertTrue(Condition := locateResult, Message := 'Did not report a locate was successful');

TEST_FINISHED();
END_METHOD

METHOD TestTryWriteBoolMethod
VAR
    jsonParser : JsonDomParser;
    jsonInitialString : T_MAXSTRING := '{"foo":"bar"}';
    newBool : BOOL := TRUE;  // Example BOOL value
    writeSuccess1 : BOOL;
    writeSuccess2 : BOOL;
    readBool1 : BOOL;
    readBool2 : BOOL;
    readResult1 : BOOL;
    readResult2 : BOOL;
    jsonOutput : T_MAXSTRING;
    expectedJsonOutput : T_MAXSTRING := '{"foo":"bar","myThing":[null,null,{"myBoolValue":true},null,true]}';
END_VAR
TEST('TestTryWriteBOOLMethod');

// @TEST-RUN
jsonParser.ParseDocument(jsonInitialString);
writeSuccess1 := jsonParser.TryWrite('.myThing[2].myBoolValue', newBool);
writeSuccess2 := jsonParser.TryWrite('.myThing[4]', newBool);
jsonOutput := jsonParser.GetDocument();

readResult1 := jsonParser.TryRead('.myThing[2].myBoolValue', readBool1);
readResult2 := jsonParser.TryRead('.myThing[4]', readBool2);
jsonParser.NewDocument();

// @TEST-ASSERT
AssertTrue(Condition := writeSuccess1, Message := 'First TryWrite operation was unsuccessful for BOOL');
AssertTrue(Condition := writeSuccess2, Message := 'Second TryWrite operation was unsuccessful for BOOL');
AssertTrue(Condition := readResult1 AND (readBool1 = newBool), Message := 'Could not read back the first written BOOL value or value mismatched');
AssertTrue(Condition := readResult2 AND (readBool2 = newBool), Message := 'Could not read back the second written BOOL value or value mismatched');
AssertEquals(Expected := expectedJsonOutput, Actual := jsonOutput, Message := 'Output JSON does not match expected for BOOL');

TEST_FINISHED();
END_METHOD

METHOD TestTryWriteDintMethod
VAR
    jsonParser : JsonDomParser;
    jsonInitialString : T_MAXSTRING := '{"foo":"bar"}';
    newDInt : DINT := -12345678;  // Example DINT value (can be negative)
    writeSuccess1 : BOOL;
    writeSuccess2 : BOOL;
    readDInt1 : DINT;
    readDInt2 : DINT;
    readResult1 : BOOL;
    readResult2 : BOOL;
    jsonOutput : T_MAXSTRING;
    expectedJsonOutput : T_MAXSTRING := '{"foo":"bar","myThing":[null,null,{"myDIntValue":-12345678},null,-12345678]}';
END_VAR
TEST('TestTryWriteDINTMethod');

// @TEST-RUN
jsonParser.ParseDocument(jsonInitialString);
writeSuccess1 := jsonParser.TryWrite('.myThing[2].myDIntValue', newDInt);
writeSuccess2 := jsonParser.TryWrite('.myThing[4]', newDInt);
jsonOutput := jsonParser.GetDocument();

readResult1 := jsonParser.TryRead('.myThing[2].myDIntValue', readDInt1);
readResult2 := jsonParser.TryRead('.myThing[4]', readDInt2);
jsonParser.NewDocument();

// @TEST-ASSERT
AssertTrue(Condition := writeSuccess1, Message := 'First TryWrite operation was unsuccessful for DINT');
AssertTrue(Condition := writeSuccess2, Message := 'Second TryWrite operation was unsuccessful for DINT');
AssertTrue(Condition := readResult1 AND (readDInt1 = newDInt), Message := 'Could not read back the first written DINT value or value mismatched');
AssertTrue(Condition := readResult2 AND (readDInt2 = newDInt), Message := 'Could not read back the second written DINT value or value mismatched');
AssertEquals(Expected := expectedJsonOutput, Actual := jsonOutput, Message := 'Output JSON does not match expected for DINT');

TEST_FINISHED();
END_METHOD

METHOD TestTryWriteIntMethod
VAR
    jsonParser : JsonDomParser;
    jsonInitialString : T_MAXSTRING := '{"foo":"bar"}';
    newInt : INT := 789;
    writeSuccess1 : BOOL;
    writeSuccess2 : BOOL;
    readInt1 : INT;
    readInt2 : INT;
    readResult1 : BOOL;
    readResult2 : BOOL;
    jsonOutput : T_MAXSTRING;
    expectedJsonOutput : T_MAXSTRING := '{"foo":"bar","myThing":[null,null,{"myIntValue":789},null,789]}';
END_VAR
TEST('TestTryWriteIntMethod');

// @TEST-RUN
jsonParser.ParseDocument(jsonInitialString);
writeSuccess1 := jsonParser.TryWrite('.myThing[2].myIntValue', newInt);
writeSuccess2 := jsonParser.TryWrite('.myThing[4]', newInt);
jsonOutput := jsonParser.GetDocument();

readResult1 := jsonParser.TryRead('.myThing[2].myIntValue', readInt1);
readResult2 := jsonParser.TryRead('.myThing[4]', readInt2);
jsonParser.NewDocument();

// @TEST-ASSERT
AssertTrue(Condition := writeSuccess1, Message := 'First TryWrite operation was unsuccessful');
AssertTrue(Condition := writeSuccess2, Message := 'Second TryWrite operation was unsuccessful');
AssertTrue(Condition := readResult1 AND (readInt1 = newInt), Message := 'Could not read back the first written INT value or value mismatched');
AssertTrue(Condition := readResult2 AND (readInt2 = newInt), Message := 'Could not read back the second written INT value or value mismatched');
AssertEquals(Expected := expectedJsonOutput, Actual := jsonOutput, Message := 'Output JSON does not match expected');

TEST_FINISHED();
END_METHOD

